LIN {X 0,Y 246.897,Z 628.128,A -85,B 0,C 180,E1 -18808.369,E2 -18808.369} C_VEL
LIN {X 0,Y 246.935,Z 628.341,A -85,B 0,C 180,E1 -18810,E2 -18810} C_VEL
LIN {X 0,Y 246.897,Z 628.119,A -85,B 0,C 180,E1 -18811.631,E2 -18811.631} C_VEL
LIN {X 0,Y 246.851,Z 627.504,A -85,B 0,C 180,E1 -18813.264,E2 -18813.264} C_VEL
LIN {X 0,Y 246.882,Z 626.502,A -85,B 0,C 180,E1 -18814.899,E2 -18814.899} C_VEL
LIN {X 0,Y 247.009,Z 625.098,A -85,B 0,C 180,E1 -18816.535,E2 -18816.535} C_VEL
LIN {X 0,Y 247.457,Z 622.154,A -85,B 0,C 180,E1 -18818.986,E2 -18818.986} C_VEL
LIN {X 0,Y 248.175,Z 618.171,A -85,B 0,C 180,E1 -18821.433,E2 -18821.433} C_VEL
LIN {X 0,Y 249.492,Z 612.051,A -85,B 0,C 180,E1 -18824.269,E2 -18824.269} C_VEL
LIN {X 0,Y 251.197,Z 605.373,A -85,B 0,C 180,E1 -18826.665,E2 -18826.665} C_VEL
LIN {X 0,Y 253.135,Z 596.963,A -85,B 0,C 180,E1 -18829.074,E2 -18829.074} C_VEL
LIN {X 0,Y 254.923,Z 588.585,A -85,B 0,C 180,E1 -18831.002,E2 -18831.002} C_VEL
LIN {X 0,Y 257.208,Z 578.088,A -85,B 0,C 180,E1 -18832.915,E2 -18832.915} C_VEL
LIN {X 0,Y 259.508,Z 566.272,A -85,B 0,C 180,E1 -18834.606,E2 -18834.606} C_VEL
LIN {X 0,Y 261.51,Z 554.368,A -85,B 0,C 180,E1 -18835.894,E2 -18835.894} C_VEL
LIN {X 0,Y 263.118,Z 541.975,A -85,B 0,C 180,E1 -18836.898,E2 -18836.898} C_VEL
LIN {X 0,Y 264.477,Z 529.21,A -85,B 0,C 180,E1 -18837.605,E2 -18837.605} C_VEL
LIN {X 0,Y 265.172,Z 515.69,A -85,B 0,C 180,E1 -18838.063,E2 -18838.063} C_VEL
LIN {X 0,Y 266.746,Z 464.43,A -85,B 0,C 180,E1 -18839.422,E2 -18839.422} C_VEL
LIN {X 0,Y 263.377,Z 442.333,A -85,B 0,C 180,E1 -18840.514,E2 -18840.514} C_VEL
LIN {X 0,Y 259.763,Z 432.973,A -85,B 0,C 180,E1 -18841.277,E2 -18841.277} C_VEL
LIN {X 0,Y 253.442,Z 418.863,A -85,B 0,C 180,E1 -18842.606,E2 -18842.606} C_VEL
LIN {X 0,Y 252.141,Z 415.736,A -85,B 0,C 180,E1 -18842.927,E2 -18842.927} C_VEL
LIN {X 0,Y 250.111,Z 407.153,A -85,B 0,C 180,E1 -18846.663,E2 -18846.663} C_VEL
LIN {X 0,Y 249.039,Z 402.966,A -85,B 0,C 180,E1 -18848.636,E2 -18848.636} C_VEL
LIN {X 0,Y 249.012,Z 402.968,A -85,B 0,C 180,E1 -18852.793,E2 -18852.793} C_VEL
LIN {X 0,Y 249.019,Z 402.965,A -85,B 0,C 180,E1 -18857.363,E2 -18857.363} C_VEL
LIN {X 0,Y 249.044,Z 402.958,A -85,B 0,C 180,E1 -18862.2,E2 -18862.2} C_VEL
LIN {X 0,Y 249.044,Z 402.958,A -85,B 0,C 180,E1 -18865.639,E2 -18865.639} C_VEL
LIN {X 0,Y 249.048,Z 402.96,A -85,B 0,C 180,E1 -18869.473,E2 -18869.473} C_VEL
LIN {X 0,Y 249.073,Z 402.959,A -85,B 0,C 180,E1 -18873.162,E2 -18873.162} C_VEL
LIN {X 0,Y 249.086,Z 402.955,A -85,B 0,C 180,E1 -18876.733,E2 -18876.733} C_VEL
LIN {X 0,Y 249.131,Z 402.949,A -85,B 0,C 180,E1 -18880.213,E2 -18880.213} C_VEL
LIN {X 0,Y 249.243,Z 402.937,A -85,B 0,C 180,E1 -18883.622,E2 -18883.622} C_VEL
LIN {X 0,Y 249.247,Z 402.936,A -85,B 0,C 180,E1 -18888.616,E2 -18888.616} C_VEL
LIN {X 0,Y 249.448,Z 402.91,A -85,B 0,C 180,E1 -18891.902,E2 -18891.902} C_VEL
LIN {X 0,Y 249.296,Z 402.924,A -85,B 0,C 180,E1 -18895.149,E2 -18895.149} C_VEL
LIN {X 0,Y 249.677,Z 402.885,A -85,B 0,C 180,E1 -18898.387,E2 -18898.387} C_VEL
LIN {X 0,Y 249.679,Z 402.876,A -85,B 0,C 180,E1 -18901.613,E2 -18901.613} C_VEL
LIN {X 0,Y 249.454,Z 402.905,A -85,B 0,C 180,E1 -18906.752,E2 -18906.752} C_VEL
LIN {X 0,Y 249.426,Z 402.916,A -85,B 0,C 180,E1 -18909.733,E2 -18909.733} C_VEL
LIN {X 0,Y 249.208,Z 402.941,A -85,B 0,C 180,E1 -18914.703,E2 -18914.703} C_VEL
LIN {X 0,Y 249.143,Z 402.948,A -85,B 0,C 180,E1 -18918.077,E2 -18918.077} C_VEL
LIN {X 0,Y 249.106,Z 402.951,A -85,B 0,C 180,E1 -18921.517,E2 -18921.517} C_VEL
LIN {X 0,Y 249.132,Z 402.951,A -85,B 0,C 180,E1 -18925.482,E2 -18925.482} C_VEL
LIN {X 0,Y 249.085,Z 402.957,A -85,B 0,C 180,E1 -18928.994,E2 -18928.994} C_VEL
LIN {X 0,Y 249.038,Z 402.962,A -85,B 0,C 180,E1 -18932.425,E2 -18932.425} C_VEL
LIN {X 0,Y 249.076,Z 402.957,A -85,B 0,C 180,E1 -18936.338,E2 -18936.338} C_VEL
LIN {X 0,Y 249.035,Z 402.96,A -85,B 0,C 180,E1 -18940.473,E2 -18940.473} C_VEL
LIN {X 0,Y 248.997,Z 402.966,A -85,B 0,C 180,E1 -18944.881,E2 -18944.881} C_VEL
LIN {X 0,Y 249.011,Z 402.965,A -85,B 0,C 180,E1 -18947.362,E2 -18947.362} C_VEL
LIN {X 0,Y 249.027,Z 402.964,A -85,B 0,C 180,E1 -18951.62,E2 -18951.62} C_VEL
LIN {X 0,Y 249.085,Z 403.063,A -85,B 0,C 180,E1 -18955.283,E2 -18955.283} C_VEL
LIN {X 0,Y 249.966,Z 406.53,A -85,B 0,C 180,E1 -18956.849,E2 -18956.849} C_VEL
LIN {X 0,Y 259.579,Z 426.19,A -85,B 0,C 180,E1 -18958.86,E2 -18958.86} C_VEL
LIN {X 0,Y 265.501,Z 440.501,A -85,B 0,C 180,E1 -18960.074,E2 -18960.074} C_VEL
LIN {X 0,Y 267.41,Z 445.672,A -85,B 0,C 180,E1 -18960.467,E2 -18960.467} C_VEL
LIN {X 0,Y 265.529,Z 503.163,A -85,B 0,C 180,E1 -18961.978,E2 -18961.978} C_VEL
LIN {X 0,Y 264.914,Z 517.263,A -85,B 0,C 180,E1 -18962.445,E2 -18962.445} C_VEL
LIN {X 0,Y 263.654,Z 530.366,A -85,B 0,C 180,E1 -18963.161,E2 -18963.161} C_VEL
LIN {X 0,Y 262.194,Z 542.855,A -85,B 0,C 180,E1 -18964.178,E2 -18964.178} C_VEL
LIN {X 0,Y 260.317,Z 554.829,A -85,B 0,C 180,E1 -18965.475,E2 -18965.475} C_VEL
LIN {X 0,Y 258.34,Z 565.491,A -85,B 0,C 180,E1 -18966.979,E2 -18966.979} C_VEL
LIN {X 0,Y 256.193,Z 576.011,A -85,B 0,C 180,E1 -18968.861,E2 -18968.861} C_VEL
LIN {X 0,Y 254.115,Z 585.636,A -85,B 0,C 180,E1 -18971.037,E2 -18971.037} C_VEL
LIN {X 0,Y 251.998,Z 593.891,A -85,B 0,C 180,E1 -18973.39,E2 -18973.39} C_VEL
LIN {X 0,Y 250.403,Z 600.535,A -85,B 0,C 180,E1 -18975.784,E2 -18975.784} C_VEL
LIN {X 0,Y 248.88,Z 606.622,A -85,B 0,C 180,E1 -18978.6,E2 -18978.6} C_VEL
LIN {X 0,Y 247.984,Z 610.573,A -85,B 0,C 180,E1 -18981.033,E2 -18981.033} C_VEL
LIN {X 0,Y 247.27,Z 614.095,A -85,B 0,C 180,E1 -18984.147,E2 -18984.147} C_VEL
LIN {X 0,Y 247.072,Z 615.873,A -85,B 0,C 180,E1 -18986.739,E2 -18986.739} C_VEL
LIN {X 0,Y 246.943,Z 616.713,A -85,B 0,C 180,E1 -18990,E2 -18990} C_VEL
LIN {X 0,Y 246.97,Z 616.519,A -85,B 0,C 180,E1 -18991.631,E2 -18991.631} C_VEL
LIN {X 0,Y 247.071,Z 615.932,A -85,B 0,C 180,E1 -18993.262,E2 -18993.262} C_VEL
LIN {X 0,Y 247.394,Z 613.607,A -85,B 0,C 180,E1 -18996.525,E2 -18996.525} C_VEL
LIN {X 0,Y 248.008,Z 610.735,A -85,B 0,C 180,E1 -18998.967,E2 -18998.967} C_VEL
LIN {X 0,Y 248.855,Z 606.842,A -85,B 0,C 180,E1 -19001.402,E2 -19001.402} C_VEL
LIN {X 0,Y 250.068,Z 601.817,A -85,B 0,C 180,E1 -19003.821,E2 -19003.821} C_VEL
LIN {X 0,Y 251.638,Z 595.488,A -85,B 0,C 180,E1 -19006.218,E2 -19006.218} C_VEL
LIN {X 0,Y 253.672,Z 587.566,A -85,B 0,C 180,E1 -19008.579,E2 -19008.579} C_VEL
LIN {X 0,Y 255.549,Z 579.262,A -85,B 0,C 180,E1 -19010.582,E2 -19010.582} C_VEL
LIN {X 0,Y 257.507,Z 569.641,A -85,B 0,C 180,E1 -19012.464,E2 -19012.464} C_VEL
LIN {X 0,Y 259.466,Z 559.937,A -85,B 0,C 180,E1 -19013.973,E2 -19013.973} C_VEL
LIN {X 0,Y 261.312,Z 549.424,A -85,B 0,C 180,E1 -19015.275,E2 -19015.275} C_VEL
LIN {X 0,Y 263.028,Z 536.765,A -85,B 0,C 180,E1 -19016.48,E2 -19016.48} C_VEL
LIN {X 0,Y 264.376,Z 524.073,A -85,B 0,C 180,E1 -19017.348,E2 -19017.348} C_VEL
LIN {X 0,Y 265.3,Z 511.903,A -85,B 0,C 180,E1 -19017.887,E2 -19017.887} C_VEL
LIN {X 0,Y 267.516,Z 446.684,A -85,B 0,C 180,E1 -19019.619,E2 -19019.619} C_VEL
LIN {X 0,Y 266.944,Z 444.324,A -85,B 0,C 180,E1 -19019.761,E2 -19019.761} C_VEL
LIN {X 0,Y 260.106,Z 427.321,A -85,B 0,C 180,E1 -19021.168,E2 -19021.168} C_VEL
LIN {X 0,Y 253.049,Z 412.735,A -85,B 0,C 180,E1 -19022.626,E2 -19022.626} C_VEL
LIN {X 0,Y 249.84,Z 406.254,A -85,B 0,C 180,E1 -19023.325,E2 -19023.325} C_VEL
LIN {X 0,Y 249.074,Z 402.959,A -85,B 0,C 180,E1 -19024.946,E2 -19024.946} C_VEL
LIN {X 0,Y 249.029,Z 402.966,A -85,B 0,C 180,E1 -19028.381,E2 -19028.381} C_VEL
LIN {X 0,Y 249.015,Z 402.965,A -85,B 0,C 180,E1 -19032.793,E2 -19032.793} C_VEL
LIN {X 0,Y 249.031,Z 402.964,A -85,B 0,C 180,E1 -19037.366,E2 -19037.366} C_VEL
LIN {X 0,Y 249.051,Z 402.951,A -85,B 0,C 180,E1 -19041.624,E2 -19041.624} C_VEL
LIN {X 0,Y 249.065,Z 402.957,A -85,B 0,C 180,E1 -19045.643,E2 -19045.643} C_VEL
LIN {X 0,Y 249.056,Z 402.959,A -85,B 0,C 180,E1 -19049.473,E2 -19049.473} C_VEL
LIN {X 0,Y 249.078,Z 402.957,A -85,B 0,C 180,E1 -19053.163,E2 -19053.163} C_VEL
LIN {X 0,Y 249.089,Z 402.957,A -85,B 0,C 180,E1 -19056.733,E2 -19056.733} C_VEL
LIN {X 0,Y 249.134,Z 402.945,A -85,B 0,C 180,E1 -19060.213,E2 -19060.213} C_VEL
LIN {X 0,Y 249.246,Z 402.938,A -85,B 0,C 180,E1 -19063.622,E2 -19063.622} C_VEL
LIN {X 0,Y 249.257,Z 402.935,A -85,B 0,C 180,E1 -19068.617,E2 -19068.617} C_VEL
LIN {X 0,Y 249.489,Z 402.9,A -85,B 0,C 180,E1 -19071.903,E2 -19071.903} C_VEL
LIN {X 0,Y 249.441,Z 402.911,A -85,B 0,C 180,E1 -19076.77,E2 -19076.77} C_VEL
LIN {X 0,Y 249.732,Z 402.87,A -85,B 0,C 180,E1 -19080,E2 -19080} C_VEL
LIN {X 0,Y 249.44,Z 402.913,A -85,B 0,C 180,E1 -19083.23,E2 -19083.23} C_VEL
LIN {X 0,Y 249.379,Z 402.913,A -85,B 0,C 180,E1 -19085.93,E2 -19085.93} C_VEL
LIN {X 0,Y 248.793,Z 402.992,A -85,B 0,C 180,E1 -19087.278,E2 -19087.278} C_VEL
LIN {X 0,Y 247.186,Z 403.196,A -85,B 0,C 180,E1 -19088.599,E2 -19088.599} C_VEL
LIN {X 0,Y 243.308,Z 403.67,A -85,B 0,C 180,E1 -19091.256,E2 -19091.256} C_VEL
LIN {X 0,Y 242.232,Z 403.806,A -85,B 0,C 180,E1 -19092.646,E2 -19092.646} C_VEL
LIN {X 0,Y 242.158,Z 403.815,A -85,B 0,C 180,E1 -19093.118,E2 -19093.118} C_VEL
LIN {X 0,Y 242.154,Z 403.814,A -85,B 0,C 180,E1 -19096.872,E2 -19096.872} C_VEL
LIN {X 0,Y 242.057,Z 403.827,A -85,B 0,C 180,E1 -19101.703,E2 -19101.703} C_VEL
LIN {X 0,Y 242.07,Z 403.831,A -85,B 0,C 180,E1 -19105.838,E2 -19105.838} C_VEL
LIN {X 0,Y 242.01,Z 403.839,A -85,B 0,C 180,E1 -19109.583,E2 -19109.583} C_VEL
LIN {X 0,Y 241.983,Z 403.842,A -85,B 0,C 180,E1 -19113.492,E2 -19113.492} C_VEL
LIN {X 0,Y 241.989,Z 403.84,A -85,B 0,C 180,E1 -19117.582,E2 -19117.582} C_VEL
LIN {X 0,Y 241.942,Z 403.847,A -85,B 0,C 180,E1 -19121.922,E2 -19121.922} C_VEL
LIN {X 0,Y 241.939,Z 403.848,A -85,B 0,C 180,E1 -19126.57,E2 -19126.57} C_VEL
LIN {X 0,Y 242.019,Z 404.013,A -85,B 0,C 180,E1 -19130.569,E2 -19130.569} C_VEL
LIN {X 0,Y 243.966,Z 411.663,A -85,B 0,C 180,E1 -19134.173,E2 -19134.173} C_VEL
LIN {X 0,Y 244.982,Z 415.904,A -85,B 0,C 180,E1 -19135.975,E2 -19135.975} C_VEL
LIN {X 0,Y 253.639,Z 434.761,A -85,B 0,C 180,E1 -19137.897,E2 -19137.897} C_VEL
LIN {X 0,Y 257.526,Z 444.708,A -85,B 0,C 180,E1 -19138.753,E2 -19138.753} C_VEL
LIN {X 0,Y 260.655,Z 464.974,A -85,B 0,C 180,E1 -19139.801,E2 -19139.801} C_VEL
LIN {X 0,Y 258.602,Z 524.234,A -85,B 0,C 180,E1 -19141.435,E2 -19141.435} C_VEL
LIN {X 0,Y 257.39,Z 537.372,A -85,B 0,C 180,E1 -19142.066,E2 -19142.066} C_VEL
LIN {X 0,Y 255.941,Z 549.464,A -85,B 0,C 180,E1 -19142.948,E2 -19142.948} C_VEL
LIN {X 0,Y 253.941,Z 561.67,A -85,B 0,C 180,E1 -19144.157,E2 -19144.157} C_VEL
LIN {X 0,Y 251.743,Z 573.234,A -85,B 0,C 180,E1 -19145.683,E2 -19145.683} C_VEL
LIN {X 0,Y 249.428,Z 583.648,A -85,B 0,C 180,E1 -19147.424,E2 -19147.424} C_VEL
LIN {X 0,Y 247.464,Z 592.165,A -85,B 0,C 180,E1 -19149.206,E2 -19149.206} C_VEL
LIN {X 0,Y 245.617,Z 600.353,A -85,B 0,C 180,E1 -19151.321,E2 -19151.321} C_VEL
LIN {X 0,Y 243.763,Z 607.705,A -85,B 0,C 180,E1 -19153.673,E2 -19153.673} C_VEL
LIN {X 0,Y 241.877,Z 614.785,A -85,B 0,C 180,E1 -19156.558,E2 -19156.558} C_VEL
LIN {X 0,Y 240.89,Z 619.5,A -85,B 0,C 180,E1 -19159.068,E2 -19159.068} C_VEL
LIN {X 0,Y 240.222,Z 623.103,A -85,B 0,C 180,E1 -19161.588,E2 -19161.588} C_VEL
LIN {X 0,Y 239.953,Z 624.961,A -85,B 0,C 180,E1 -19163.272,E2 -19163.272} C_VEL
LIN {X 0,Y 239.755,Z 627.352,A -85,B 0,C 180,E1 -19166.639,E2 -19166.639} C_VEL
LIN {X 0,Y 239.809,Z 627.961,A -85,B 0,C 180,E1 -19168.32,E2 -19168.32} C_VEL
LIN {X 0,Y 239.846,Z 628.174,A -85,B 0,C 180,E1 -19170,E2 -19170} C_VEL
LIN {X 0,Y 239.809,Z 627.951,A -85,B 0,C 180,E1 -19171.679,E2 -19171.679} C_VEL
LIN {X 0,Y 239.771,Z 626.542,A -85,B 0,C 180,E1 -19174.736,E2 -19174.736} C_VEL
LIN {X 0,Y 239.952,Z 624.93,A -85,B 0,C 180,E1 -19176.728,E2 -19176.728} C_VEL
LIN {X 0,Y 240.416,Z 621.985,A -85,B 0,C 180,E1 -19179.252,E2 -19179.252} C_VEL
LIN {X 0,Y 241.198,Z 618.003,A -85,B 0,C 180,E1 -19181.769,E2 -19181.769} C_VEL
LIN {X 0,Y 242.611,Z 611.882,A -85,B 0,C 180,E1 -19184.683,E2 -19184.683} C_VEL
LIN {X 0,Y 244.359,Z 605.203,A -85,B 0,C 180,E1 -19187.145,E2 -19187.145} C_VEL
LIN {X 0,Y 246.242,Z 597.458,A -85,B 0,C 180,E1 -19189.436,E2 -19189.436} C_VEL
LIN {X 0,Y 248.275,Z 588.414,A -85,B 0,C 180,E1 -19191.592,E2 -19191.592} C_VEL
LIN {X 0,Y 250.665,Z 577.917,A -85,B 0,C 180,E1 -19193.549,E2 -19193.549} C_VEL
LIN {X 0,Y 253.059,Z 566.1,A -85,B 0,C 180,E1 -19195.277,E2 -19195.277} C_VEL
LIN {X 0,Y 255.149,Z 554.195,A -85,B 0,C 180,E1 -19196.59,E2 -19196.59} C_VEL
LIN {X 0,Y 256.823,Z 541.801,A -85,B 0,C 180,E1 -19197.613,E2 -19197.613} C_VEL
LIN {X 0,Y 258.22,Z 529.031,A -85,B 0,C 180,E1 -19198.333,E2 -19198.333} C_VEL
LIN {X 0,Y 258.939,Z 515.502,A -85,B 0,C 180,E1 -19198.8,E2 -19198.8} C_VEL
LIN {X 0,Y 260.581,Z 465.599,A -85,B 0,C 180,E1 -19200.147,E2 -19200.147} C_VEL
LIN {X 0,Y 257.439,Z 444.492,A -85,B 0,C 180,E1 -19201.222,E2 -19201.222} C_VEL
LIN {X 0,Y 251.429,Z 429.81,A -85,B 0,C 180,E1 -19202.534,E2 -19202.534} C_VEL
LIN {X 0,Y 246.214,Z 418.717,A -85,B 0,C 180,E1 -19203.685,E2 -19203.685} C_VEL
LIN {X 0,Y 244.856,Z 415.514,A -85,B 0,C 180,E1 -19204.047,E2 -19204.047} C_VEL
LIN {X 0,Y 242.907,Z 407.421,A -85,B 0,C 180,E1 -19207.738,E2 -19207.738} C_VEL
LIN {X 0,Y 241.986,Z 403.841,A -85,B 0,C 180,E1 -19209.531,E2 -19209.531} C_VEL
LIN {X 0,Y 241.935,Z 403.845,A -85,B 0,C 180,E1 -19214.201,E2 -19214.201} C_VEL
LIN {X 0,Y 241.94,Z 403.846,A -85,B 0,C 180,E1 -19218.078,E2 -19218.078} C_VEL
LIN {X 0,Y 241.99,Z 403.836,A -85,B 0,C 180,E1 -19222.418,E2 -19222.418} C_VEL
LIN {X 0,Y 241.981,Z 403.841,A -85,B 0,C 180,E1 -19226.507,E2 -19226.507} C_VEL
LIN {X 0,Y 242.014,Z 403.84,A -85,B 0,C 180,E1 -19230.597,E2 -19230.597} C_VEL
LIN {X 0,Y 242.069,Z 403.832,A -85,B 0,C 180,E1 -19234.183,E2 -19234.183} C_VEL
LIN {X 0,Y 242.066,Z 403.833,A -85,B 0,C 180,E1 -19238.29,E2 -19238.29} C_VEL
LIN {X 0,Y 242.164,Z 403.819,A -85,B 0,C 180,E1 -19243.278,E2 -19243.278} C_VEL
LIN {X 0,Y 242.183,Z 403.819,A -85,B 0,C 180,E1 -19248.28,E2 -19248.28} C_VEL
LIN {X 0,Y 242.395,Z 403.788,A -85,B 0,C 180,E1 -19251.665,E2 -19251.665} C_VEL
LIN {X 0,Y 242.257,Z 403.801,A -85,B 0,C 180,E1 -19255.007,E2 -19255.007} C_VEL
LIN {X 0,Y 242.638,Z 403.762,A -85,B 0,C 180,E1 -19258.34,E2 -19258.34} C_VEL
LIN {X 0,Y 242.639,Z 403.753,A -85,B 0,C 180,E1 -19261.66,E2 -19261.66} C_VEL
LIN {X 0,Y 242.432,Z 403.78,A -85,B 0,C 180,E1 -19266.731,E2 -19266.731} C_VEL
LIN {X 0,Y 242.347,Z 403.797,A -85,B 0,C 180,E1 -19270.02,E2 -19270.02} C_VEL
LIN {X 0,Y 242.169,Z 403.818,A -85,B 0,C 180,E1 -19275.141,E2 -19275.141} C_VEL
LIN {X 0,Y 242.082,Z 403.829,A -85,B 0,C 180,E1 -19278.624,E2 -19278.624} C_VEL
LIN {X 0,Y 242.052,Z 403.83,A -85,B 0,C 180,E1 -19282.176,E2 -19282.176} C_VEL
LIN {X 0,Y 242.068,Z 403.828,A -85,B 0,C 180,E1 -19285.838,E2 -19285.838} C_VEL
LIN {X 0,Y 242.032,Z 403.834,A -85,B 0,C 180,E1 -19289.58,E2 -19289.58} C_VEL
LIN {X 0,Y 241.993,Z 403.839,A -85,B 0,C 180,E1 -19293.491,E2 -19293.491} C_VEL
LIN {X 0,Y 242.012,Z 403.835,A -85,B 0,C 180,E1 -19297.578,E2 -19297.578} C_VEL
LIN {X 0,Y 241.95,Z 403.846,A -85,B 0,C 180,E1 -19301.92,E2 -19301.92} C_VEL
LIN {X 0,Y 241.928,Z 403.847,A -85,B 0,C 180,E1 -19306.573,E2 -19306.573} C_VEL
LIN {X 0,Y 241.958,Z 403.846,A -85,B 0,C 180,E1 -19310.281,E2 -19310.281} C_VEL
LIN {X 0,Y 242.03,Z 403.853,A -85,B 0,C 180,E1 -19314.396,E2 -19314.396} C_VEL
LIN {X 0,Y 242.707,Z 406.604,A -85,B 0,C 180,E1 -19315.716,E2 -19315.716} C_VEL
LIN {X 0,Y 251.706,Z 424.526,A -85,B 0,C 180,E1 -19317.707,E2 -19317.707} C_VEL
LIN {X 0,Y 257.992,Z 438.988,A -85,B 0,C 180,E1 -19319.053,E2 -19319.053} C_VEL
LIN {X 0,Y 261.168,Z 447.286,A -85,B 0,C 180,E1 -19319.733,E2 -19319.733} C_VEL
LIN {X 0,Y 259.33,Z 502.465,A -85,B 0,C 180,E1 -19321.219,E2 -19321.219} C_VEL
LIN {X 0,Y 258.621,Z 517.764,A -85,B 0,C 180,E1 -19321.73,E2 -19321.73} C_VEL
LIN {X 0,Y 257.351,Z 530.542,A -85,B 0,C 180,E1 -19322.449,E2 -19322.449} C_VEL
LIN {X 0,Y 255.835,Z 543.028,A -85,B 0,C 180,E1 -19323.487,E2 -19323.487} C_VEL
LIN {X 0,Y 253.894,Z 555.001,A -85,B 0,C 180,E1 -19324.812,E2 -19324.812} C_VEL
LIN {X 0,Y 251.82,Z 565.662,A -85,B 0,C 180,E1 -19326.348,E2 -19326.348} C_VEL
LIN {X 0,Y 249.461,Z 576.75,A -85,B 0,C 180,E1 -19328.389,E2 -19328.389} C_VEL
LIN {X 0,Y 247.413,Z 585.805,A -85,B 0,C 180,E1 -19330.502,E2 -19330.502} C_VEL
LIN {X 0,Y 245.206,Z 594.06,A -85,B 0,C 180,E1 -19332.916,E2 -19332.916} C_VEL
LIN {X 0,Y 243.523,Z 600.704,A -85,B 0,C 180,E1 -19335.373,E2 -19335.373} C_VEL
LIN {X 0,Y 241.921,Z 606.791,A -85,B 0,C 180,E1 -19338.267,E2 -19338.267} C_VEL
LIN {X 0,Y 240.972,Z 610.741,A -85,B 0,C 180,E1 -19340.77,E2 -19340.77} C_VEL
LIN {X 0,Y 240.171,Z 614.479,A -85,B 0,C 180,E1 -19344.227,E2 -19344.227} C_VEL
LIN {X 0,Y 239.995,Z 616.04,A -85,B 0,C 180,E1 -19346.643,E2 -19346.643} C_VEL
LIN {X 0,Y 239.885,Z 616.65,A -85,B 0,C 180,E1 -19348.321,E2 -19348.321} C_VEL
LIN {X 0,Y 239.854,Z 616.88,A -85,B 0,C 180,E1 -19350,E2 -19350} C_VEL
LIN {X 0,Y 239.885,Z 616.686,A -85,B 0,C 180,E1 -19351.679,E2 -19351.679} C_VEL
LIN {X 0,Y 239.994,Z 616.099,A -85,B 0,C 180,E1 -19353.358,E2 -19353.358} C_VEL
LIN {X 0,Y 240.349,Z 613.773,A -85,B 0,C 180,E1 -19356.717,E2 -19356.717} C_VEL
LIN {X 0,Y 240.988,Z 610.902,A -85,B 0,C 180,E1 -19359.23,E2 -19359.23} C_VEL
LIN {X 0,Y 241.893,Z 607.008,A -85,B 0,C 180,E1 -19361.735,E2 -19361.735} C_VEL
LIN {X 0,Y 243.176,Z 601.983,A -85,B 0,C 180,E1 -19364.221,E2 -19364.221} C_VEL
LIN {X 0,Y 244.825,Z 595.654,A -85,B 0,C 180,E1 -19366.683,E2 -19366.683} C_VEL
LIN {X 0,Y 246.957,Z 587.731,A -85,B 0,C 180,E1 -19369.104,E2 -19369.104} C_VEL
LIN {X 0,Y 248.766,Z 580.035,A -85,B 0,C 180,E1 -19371.021,E2 -19371.021} C_VEL
LIN {X 0,Y 250.962,Z 569.804,A -85,B 0,C 180,E1 -19373.083,E2 -19373.083} C_VEL
LIN {X 0,Y 253.282,Z 558.705,A -85,B 0,C 180,E1 -19374.815,E2 -19374.815} C_VEL
LIN {X 0,Y 255.181,Z 547.823,A -85,B 0,C 180,E1 -19376.146,E2 -19376.146} C_VEL
LIN {X 0,Y 256.851,Z 535.797,A -85,B 0,C 180,E1 -19377.279,E2 -19377.279} C_VEL
LIN {X 0,Y 258.152,Z 523.418,A -85,B 0,C 180,E1 -19378.121,E2 -19378.121} C_VEL
LIN {X 0,Y 259.07,Z 510.548,A -85,B 0,C 180,E1 -19378.674,E2 -19378.674} C_VEL
LIN {X 0,Y 259.842,Z 490.019,A -85,B 0,C 180,E1 -19379.236,E2 -19379.236} C_VEL
LIN {X 0,Y 261.259,Z 447.451,A -85,B 0,C 180,E1 -19380.383,E2 -19380.383} C_VEL
LIN {X 0,Y 255.083,Z 431.858,A -85,B 0,C 180,E1 -19381.709,E2 -19381.709} C_VEL
LIN {X 0,Y 248.25,Z 417.405,A -85,B 0,C 180,E1 -19383.183,E2 -19383.183} C_VEL
LIN {X 0,Y 242.656,Z 406.378,A -85,B 0,C 180,E1 -19384.479,E2 -19384.479} C_VEL
LIN {X 0,Y 242.009,Z 403.833,A -85,B 0,C 180,E1 -19385.808,E2 -19385.808} C_VEL
LIN {X 0,Y 241.959,Z 403.846,A -85,B 0,C 180,E1 -19389.719,E2 -19389.719} C_VEL
LIN {X 0,Y 241.939,Z 403.848,A -85,B 0,C 180,E1 -19394.201,E2 -19394.201} C_VEL
LIN {X 0,Y 241.956,Z 403.844,A -85,B 0,C 180,E1 -19398.081,E2 -19398.081} C_VEL
LIN {X 0,Y 242.014,Z 403.831,A -85,B 0,C 180,E1 -19402.422,E2 -19402.422} C_VEL
LIN {X 0,Y 241.995,Z 403.837,A -85,B 0,C 180,E1 -19406.509,E2 -19406.509} C_VEL
LIN {X 0,Y 242.041,Z 403.83,A -85,B 0,C 180,E1 -19410.587,E2 -19410.587} C_VEL
LIN {X 0,Y 242.071,Z 403.827,A -85,B 0,C 180,E1 -19414.183,E2 -19414.183} C_VEL
LIN {X 0,Y 242.069,Z 403.832,A -85,B 0,C 180,E1 -19418.29,E2 -19418.29} C_VEL
LIN {X 0,Y 242.167,Z 403.818,A -85,B 0,C 180,E1 -19423.278,E2 -19423.278} C_VEL
LIN {X 0,Y 242.191,Z 403.815,A -85,B 0,C 180,E1 -19428.28,E2 -19428.28} C_VEL
LIN {X 0,Y 242.44,Z 403.78,A -85,B 0,C 180,E1 -19431.666,E2 -19431.666} C_VEL
LIN {X 0,Y 242.266,Z 403.805,A -85,B 0,C 180,E1 -19435.007,E2 -19435.007} C_VEL
LIN {X 0,Y 242.641,Z 403.751,A -85,B 0,C 180,E1 -19438.34,E2 -19438.34} C_VEL
LIN {X 0,Y 242.641,Z 403.76,A -85,B 0,C 180,E1 -19441.66,E2 -19441.66} C_VEL
LIN {X 0,Y 242.422,Z 403.782,A -85,B 0,C 180,E1 -19446.659,E2 -19446.659} C_VEL
LIN {X 0,Y 242.271,Z 403.802,A -85,B 0,C 180,E1 -19450.023,E2 -19450.023} C_VEL
LIN {X 0,Y 242.158,Z 403.815,A -85,B 0,C 180,E1 -19453.118,E2 -19453.118} C_VEL
LIN {X 0,Y 241.506,Z 403.904,A -85,B 0,C 180,E1 -19454.506,E2 -19454.506} C_VEL
LIN {X 0,Y 238.588,Z 404.266,A -85,B 0,C 180,E1 -19456.766,E2 -19456.766} C_VEL
LIN {X 0,Y 236.104,Z 404.571,A -85,B 0,C 180,E1 -19458.609,E2 -19458.609} C_VEL
LIN {X 0,Y 235.062,Z 404.704,A -85,B 0,C 180,E1 -19460.041,E2 -19460.041} C_VEL
LIN {X 0,Y 234.991,Z 404.71,A -85,B 0,C 180,E1 -19460.527,E2 -19460.527} C_VEL
LIN {X 0,Y 234.991,Z 404.713,A -85,B 0,C 180,E1 -19464.753,E2 -19464.753} C_VEL
LIN {X 0,Y 234.94,Z 404.717,A -85,B 0,C 180,E1 -19468.596,E2 -19468.596} C_VEL
LIN {X 0,Y 234.946,Z 404.718,A -85,B 0,C 180,E1 -19473.114,E2 -19473.114} C_VEL
LIN {X 0,Y 234.928,Z 404.719,A -85,B 0,C 180,E1 -19476.749,E2 -19476.749} C_VEL
LIN {X 0,Y 234.944,Z 404.718,A -85,B 0,C 180,E1 -19478.944,E2 -19478.944} C_VEL
LIN {X 0,Y 234.892,Z 404.726,A -85,B 0,C 180,E1 -19483.485,E2 -19483.485} C_VEL
LIN {X 0,Y 234.892,Z 404.726,A -85,B 0,C 180,E1 -19486.514,E2 -19486.514} C_VEL
LIN {X 0,Y 234.923,Z 404.875,A -85,B 0,C 180,E1 -19489.619,E2 -19489.619} C_VEL
LIN {X 0,Y 237.05,Z 413.026,A -85,B 0,C 180,E1 -19493.632,E2 -19493.632} C_VEL
LIN {X 0,Y 237.559,Z 415.398,A -85,B 0,C 180,E1 -19494.734,E2 -19494.734} C_VEL
LIN {X 0,Y 239.563,Z 419.492,A -85,B 0,C 180,E1 -19495.228,E2 -19495.228} C_VEL
LIN {X 0,Y 247.265,Z 436.042,A -85,B 0,C 180,E1 -19497.014,E2 -19497.014} C_VEL
LIN {X 0,Y 251.734,Z 447.593,A -85,B 0,C 180,E1 -19498.049,E2 -19498.049} C_VEL
LIN {X 0,Y 254.565,Z 466.785,A -85,B 0,C 180,E1 -19499.063,E2 -19499.063} C_VEL
LIN {X 0,Y 252.388,Z 524.081,A -85,B 0,C 180,E1 -19500.664,E2 -19500.664} C_VEL
LIN {X 0,Y 251.157,Z 537.215,A -85,B 0,C 180,E1 -19501.309,E2 -19501.309} C_VEL
LIN {X 0,Y 249.643,Z 549.304,A -85,B 0,C 180,E1 -19502.207,E2 -19502.207} C_VEL
LIN {X 0,Y 247.574,Z 561.507,A -85,B 0,C 180,E1 -19503.441,E2 -19503.441} C_VEL
LIN {X 0,Y 245.257,Z 573.07,A -85,B 0,C 180,E1 -19504.996,E2 -19504.996} C_VEL
LIN {X 0,Y 242.889,Z 583.484,A -85,B 0,C 180,E1 -19506.781,E2 -19506.781} C_VEL
LIN {X 0,Y 240.812,Z 592,A -85,B 0,C 180,E1 -19508.604,E2 -19508.604} C_VEL
LIN {X 0,Y 239.019,Z 599.673,A -85,B 0,C 180,E1 -19510.625,E2 -19510.625} C_VEL
LIN {X 0,Y 236.94,Z 607.539,A -85,B 0,C 180,E1 -19513.19,E2 -19513.19} C_VEL
LIN {X 0,Y 234.938,Z 614.618,A -85,B 0,C 180,E1 -19516.154,E2 -19516.154} C_VEL
LIN {X 0,Y 233.905,Z 619.333,A -85,B 0,C 180,E1 -19518.737,E2 -19518.737} C_VEL
LIN {X 0,Y 233.191,Z 622.936,A -85,B 0,C 180,E1 -19521.333,E2 -19521.333} C_VEL
LIN {X 0,Y 232.89,Z 624.795,A -85,B 0,C 180,E1 -19523.067,E2 -19523.067} C_VEL
LIN {X 0,Y 232.664,Z 627.185,A -85,B 0,C 180,E1 -19526.536,E2 -19526.536} C_VEL
LIN {X 0,Y 232.722,Z 627.795,A -85,B 0,C 180,E1 -19528.269,E2 -19528.269} C_VEL
LIN {X 0,Y 232.759,Z 628.008,A -85,B 0,C 180,E1 -19530,E2 -19530} C_VEL
LIN {X 0,Y 232.722,Z 627.784,A -85,B 0,C 180,E1 -19531.73,E2 -19531.73} C_VEL
LIN {X 0,Y 232.731,Z 626.167,A -85,B 0,C 180,E1 -19535.197,E2 -19535.197} C_VEL
LIN {X 0,Y 232.89,Z 624.762,A -85,B 0,C 180,E1 -19536.933,E2 -19536.933} C_VEL
LIN {X 0,Y 233.395,Z 621.817,A -85,B 0,C 180,E1 -19539.533,E2 -19539.533} C_VEL
LIN {X 0,Y 234.231,Z 617.834,A -85,B 0,C 180,E1 -19542.124,E2 -19542.124} C_VEL
LIN {X 0,Y 235.736,Z 611.713,A -85,B 0,C 180,E1 -19545.121,E2 -19545.121} C_VEL
LIN {X 0,Y 237.519,Z 605.033,A -85,B 0,C 180,E1 -19547.655,E2 -19547.655} C_VEL
LIN {X 0,Y 239.365,Z 597.938,A -85,B 0,C 180,E1 -19549.823,E2 -19549.823} C_VEL
LIN {X 0,Y 241.667,Z 588.244,A -85,B 0,C 180,E1 -19552.213,E2 -19552.213} C_VEL
LIN {X 0,Y 244.172,Z 577.746,A -85,B 0,C 180,E1 -19554.215,E2 -19554.215} C_VEL
LIN {X 0,Y 246.658,Z 565.928,A -85,B 0,C 180,E1 -19555.981,E2 -19555.981} C_VEL
LIN {X 0,Y 248.823,Z 554.022,A -85,B 0,C 180,E1 -19557.321,E2 -19557.321} C_VEL
LIN {X 0,Y 250.38,Z 542.927,A -85,B 0,C 180,E1 -19558.273,E2 -19558.273} C_VEL
LIN {X 0,Y 251.928,Z 529.783,A -85,B 0,C 180,E1 -19559.05,E2 -19559.05} C_VEL
LIN {X 0,Y 252.687,Z 517.104,A -85,B 0,C 180,E1 -19559.525,E2 -19559.525} C_VEL
LIN {X 0,Y 254.357,Z 465.807,A -85,B 0,C 180,E1 -19560.952,E2 -19560.952} C_VEL
LIN {X 0,Y 251.523,Z 446.656,A -85,B 0,C 180,E1 -19561.965,E2 -19561.965} C_VEL
LIN {X 0,Y 244.883,Z 430.758,A -85,B 0,C 180,E1 -19563.477,E2 -19563.477} C_VEL
LIN {X 0,Y 239.172,Z 418.866,A -85,B 0,C 180,E1 -19564.804,E2 -19564.804} C_VEL
LIN {X 0,Y 237.555,Z 415.333,A -85,B 0,C 180,E1 -19565.237,E2 -19565.237} C_VEL
LIN {X 0,Y 235.776,Z 407.971,A -85,B 0,C 180,E1 -19568.753,E2 -19568.753} C_VEL
LIN {X 0,Y 234.913,Z 404.724,A -85,B 0,C 180,E1 -19570.453,E2 -19570.453} C_VEL
LIN {X 0,Y 234.899,Z 404.721,A -85,B 0,C 180,E1 -19574.105,E2 -19574.105} C_VEL
LIN {X 0,Y 234.885,Z 404.722,A -85,B 0,C 180,E1 -19578.832,E2 -19578.832} C_VEL
LIN {X 0,Y 234.919,Z 404.72,A -85,B 0,C 180,E1 -19581.079,E2 -19581.079} C_VEL
LIN {X 0,Y 234.931,Z 404.716,A -85,B 0,C 180,E1 -19585.362,E2 -19585.362} C_VEL
LIN {X 0,Y 234.923,Z 404.72,A -85,B 0,C 180,E1 -19589.431,E2 -19589.431} C_VEL
LIN {X 0,Y 234.995,Z 404.712,A -85,B 0,C 180,E1 -19593.794,E2 -19593.794} C_VEL
LIN {X 0,Y 235.029,Z 404.708,A -85,B 0,C 180,E1 -19598.971,E2 -19598.971} C_VEL
LIN {X 0,Y 235.098,Z 404.699,A -85,B 0,C 180,E1 -19603.059,E2 -19603.059} C_VEL
LIN {X 0,Y 235.117,Z 404.698,A -85,B 0,C 180,E1 -19607.922,E2 -19607.922} C_VEL
LIN {X 0,Y 235.328,Z 404.667,A -85,B 0,C 180,E1 -19611.412,E2 -19611.412} C_VEL
LIN {X 0,Y 235.37,Z 404.665,A -85,B 0,C 180,E1 -19613.14,E2 -19613.14} C_VEL
LIN {X 0,Y 235.597,Z 404.64,A -85,B 0,C 180,E1 -19618.291,E2 -19618.291} C_VEL
LIN {X 0,Y 235.599,Z 404.63,A -85,B 0,C 180,E1 -19621.709,E2 -19621.709} C_VEL
LIN {X 0,Y 235.408,Z 404.655,A -85,B 0,C 180,E1 -19626.859,E2 -19626.859} C_VEL
LIN {X 0,Y 235.255,Z 404.678,A -85,B 0,C 180,E1 -19630.326,E2 -19630.326} C_VEL
LIN {X 0,Y 235.116,Z 404.697,A -85,B 0,C 180,E1 -19635.606,E2 -19635.606} C_VEL
LIN {X 0,Y 235.022,Z 404.709,A -85,B 0,C 180,E1 -19639.205,E2 -19639.205} C_VEL
LIN {X 0,Y 234.983,Z 404.712,A -85,B 0,C 180,E1 -19642.881,E2 -19642.881} C_VEL
LIN {X 0,Y 234.971,Z 404.712,A -85,B 0,C 180,E1 -19646.657,E2 -19646.657} C_VEL
LIN {X 0,Y 234.934,Z 404.716,A -85,B 0,C 180,E1 -19650.568,E2 -19650.568} C_VEL
LIN {X 0,Y 234.962,Z 404.713,A -85,B 0,C 180,E1 -19654.633,E2 -19654.633} C_VEL
LIN {X 0,Y 234.943,Z 404.717,A -85,B 0,C 180,E1 -19658.945,E2 -19658.945} C_VEL
LIN {X 0,Y 234.889,Z 404.724,A -85,B 0,C 180,E1 -19663.486,E2 -19663.486} C_VEL
LIN {X 0,Y 234.881,Z 404.725,A -85,B 0,C 180,E1 -19666.513,E2 -19666.513} C_VEL
LIN {X 0,Y 234.92,Z 404.723,A -85,B 0,C 180,E1 -19671.079,E2 -19671.079} C_VEL
LIN {X 0,Y 235,Z 404.854,A -85,B 0,C 180,E1 -19673.546,E2 -19673.546} C_VEL
LIN {X 0,Y 235.464,Z 406.711,A -85,B 0,C 180,E1 -19674.501,E2 -19674.501} C_VEL
LIN {X 0,Y 244.565,Z 424.453,A -85,B 0,C 180,E1 -19676.633,E2 -19676.633} C_VEL
LIN {X 0,Y 251.701,Z 440.296,A -85,B 0,C 180,E1 -19678.227,E2 -19678.227} C_VEL
LIN {X 0,Y 255.022,Z 449.005,A -85,B 0,C 180,E1 -19678.973,E2 -19678.973} C_VEL
LIN {X 0,Y 253.073,Z 503.916,A -85,B 0,C 180,E1 -19680.479,E2 -19680.479} C_VEL
LIN {X 0,Y 252.344,Z 518.361,A -85,B 0,C 180,E1 -19680.984,E2 -19680.984} C_VEL
LIN {X 0,Y 251.084,Z 530.718,A -85,B 0,C 180,E1 -19681.7,E2 -19681.7} C_VEL
LIN {X 0,Y 249.511,Z 543.202,A -85,B 0,C 180,E1 -19682.76,E2 -19682.76} C_VEL
LIN {X 0,Y 247.502,Z 555.172,A -85,B 0,C 180,E1 -19684.114,E2 -19684.114} C_VEL
LIN {X 0,Y 245.351,Z 565.833,A -85,B 0,C 180,E1 -19685.684,E2 -19685.684} C_VEL
LIN {X 0,Y 243.2,Z 575.546,A -85,B 0,C 180,E1 -19687.487,E2 -19687.487} C_VEL
LIN {X 0,Y 241.129,Z 584.38,A -85,B 0,C 180,E1 -19689.528,E2 -19689.528} C_VEL
LIN {X 0,Y 238.823,Z 593,A -85,B 0,C 180,E1 -19692.002,E2 -19692.002} C_VEL
LIN {X 0,Y 236.884,Z 599.872,A -85,B 0,C 180,E1 -19694.513,E2 -19694.513} C_VEL
LIN {X 0,Y 235.376,Z 605.372,A -85,B 0,C 180,E1 -19697.06,E2 -19697.06} C_VEL
LIN {X 0,Y 234.242,Z 609.687,A -85,B 0,C 180,E1 -19699.629,E2 -19699.629} C_VEL
LIN {X 0,Y 233.716,Z 611.969,A -85,B 0,C 180,E1 -19701.353,E2 -19701.353} C_VEL
LIN {X 0,Y 233.094,Z 614.82,A -85,B 0,C 180,E1 -19704.26,E2 -19704.26} C_VEL
LIN {X 0,Y 232.9,Z 616.208,A -85,B 0,C 180,E1 -19706.54,E2 -19706.54} C_VEL
LIN {X 0,Y 232.802,Z 616.817,A -85,B 0,C 180,E1 -19708.27,E2 -19708.27} C_VEL
LIN {X 0,Y 232.768,Z 617.047,A -85,B 0,C 180,E1 -19710,E2 -19710} C_VEL
LIN {X 0,Y 232.802,Z 616.853,A -85,B 0,C 180,E1 -19711.73,E2 -19711.73} C_VEL
LIN {X 0,Y 232.899,Z 616.266,A -85,B 0,C 180,E1 -19713.46,E2 -19713.46} C_VEL
LIN {X 0,Y 233.3,Z 613.94,A -85,B 0,C 180,E1 -19716.921,E2 -19716.921} C_VEL
LIN {X 0,Y 233.989,Z 611.068,A -85,B 0,C 180,E1 -19719.509,E2 -19719.509} C_VEL
LIN {X 0,Y 234.946,Z 607.174,A -85,B 0,C 180,E1 -19722.087,E2 -19722.087} C_VEL
LIN {X 0,Y 236.299,Z 602.149,A -85,B 0,C 180,E1 -19724.644,E2 -19724.644} C_VEL
LIN {X 0,Y 238.035,Z 595.819,A -85,B 0,C 180,E1 -19727.173,E2 -19727.173} C_VEL
LIN {X 0,Y 240.265,Z 587.895,A -85,B 0,C 180,E1 -19729.657,E2 -19729.657} C_VEL
LIN {X 0,Y 242.462,Z 578.816,A -85,B 0,C 180,E1 -19731.943,E2 -19731.943} C_VEL
LIN {X 0,Y 244.686,Z 568.868,A -85,B 0,C 180,E1 -19733.936,E2 -19733.936} C_VEL
LIN {X 0,Y 247.109,Z 557.445,A -85,B 0,C 180,E1 -19735.705,E2 -19735.705} C_VEL
LIN {X 0,Y 249.118,Z 546.223,A -85,B 0,C 180,E1 -19737.06,E2 -19737.06} C_VEL
LIN {X 0,Y 250.75,Z 534.818,A -85,B 0,C 180,E1 -19738.114,E2 -19738.114} C_VEL
LIN {X 0,Y 252.086,Z 521.75,A -85,B 0,C 180,E1 -19738.974,E2 -19738.974} C_VEL
LIN {X 0,Y 252.948,Z 509.19,A -85,B 0,C 180,E1 -19739.493,E2 -19739.493} C_VEL
LIN {X 0,Y 253.691,Z 490.209,A -85,B 0,C 180,E1 -19740.015,E2 -19740.015} C_VEL
LIN {X 0,Y 255.123,Z 449.136,A -85,B 0,C 180,E1 -19741.144,E2 -19741.144} C_VEL
LIN {X 0,Y 248.838,Z 433.456,A -85,B 0,C 180,E1 -19742.553,E2 -19742.553} C_VEL
LIN {X 0,Y 241.01,Z 417.344,A -85,B 0,C 180,E1 -19744.324,E2 -19744.324} C_VEL
LIN {X 0,Y 236.78,Z 409.483,A -85,B 0,C 180,E1 -19745.316,E2 -19745.316} C_VEL
LIN {X 0,Y 235.428,Z 406.64,A -85,B 0,C 180,E1 -19745.667,E2 -19745.667} C_VEL
LIN {X 0,Y 234.97,Z 404.71,A -85,B 0,C 180,E1 -19746.742,E2 -19746.742} C_VEL
LIN {X 0,Y 234.887,Z 404.725,A -85,B 0,C 180,E1 -19751.168,E2 -19751.168} C_VEL
LIN {X 0,Y 234.905,Z 404.721,A -85,B 0,C 180,E1 -19755.894,E2 -19755.894} C_VEL
LIN {X 0,Y 234.909,Z 404.715,A -85,B 0,C 180,E1 -19758.837,E2 -19758.837} C_VEL
LIN {X 0,Y 234.958,Z 404.699,A -85,B 0,C 180,E1 -19761.086,E2 -19761.086} C_VEL
LIN {X 0,Y 234.964,Z 404.713,A -85,B 0,C 180,E1 -19765.367,E2 -19765.367} C_VEL
LIN {X 0,Y 234.973,Z 404.71,A -85,B 0,C 180,E1 -19770.157,E2 -19770.157} C_VEL
LIN {X 0,Y 234.998,Z 404.712,A -85,B 0,C 180,E1 -19773.794,E2 -19773.794} C_VEL
LIN {X 0,Y 235.032,Z 404.705,A -85,B 0,C 180,E1 -19778.972,E2 -19778.972} C_VEL
LIN {X 0,Y 235.101,Z 404.699,A -85,B 0,C 180,E1 -19783.059,E2 -19783.059} C_VEL
LIN {X 0,Y 235.151,Z 404.688,A -85,B 0,C 180,E1 -19787.924,E2 -19787.924} C_VEL
LIN {X 0,Y 235.395,Z 404.659,A -85,B 0,C 180,E1 -19791.415,E2 -19791.415} C_VEL
LIN {X 0,Y 235.411,Z 404.65,A -85,B 0,C 180,E1 -19793.141,E2 -19793.141} C_VEL
LIN {X 0,Y 235.601,Z 404.628,A -85,B 0,C 180,E1 -19798.291,E2 -19798.291} C_VEL
LIN {X 0,Y 235.6,Z 404.637,A -85,B 0,C 180,E1 -19801.709,E2 -19801.709} C_VEL
LIN {X 0,Y 235.373,Z 404.66,A -85,B 0,C 180,E1 -19806.86,E2 -19806.86} C_VEL
LIN {X 0,Y 235.218,Z 404.679,A -85,B 0,C 180,E1 -19810.327,E2 -19810.327} C_VEL
LIN {X 0,Y 235.118,Z 404.695,A -85,B 0,C 180,E1 -19815.606,E2 -19815.606} C_VEL
LIN {X 0,Y 235.013,Z 404.709,A -85,B 0,C 180,E1 -19819.205,E2 -19819.205} C_VEL
LIN {X 0,Y 234.991,Z 404.71,A -85,B 0,C 180,E1 -19820.527,E2 -19820.527} C_VEL
LIN {X 0,Y 234.353,Z 404.794,A -85,B 0,C 180,E1 -19821.958,E2 -19821.958} C_VEL
LIN {X 0,Y 231.483,Z 405.155,A -85,B 0,C 180,E1 -19824.291,E2 -19824.291} C_VEL
LIN {X 0,Y 229.016,Z 405.46,A -85,B 0,C 180,E1 -19826.194,E2 -19826.194} C_VEL
LIN {X 0,Y 227.95,Z 405.589,A -85,B 0,C 180,E1 -19827.672,E2 -19827.672} C_VEL
LIN {X 0,Y 227.86,Z 405.598,A -85,B 0,C 180,E1 -19828.174,E2 -19828.174} C_VEL
LIN {X 0,Y 227.87,Z 405.6,A -85,B 0,C 180,E1 -19831.622,E2 -19831.622} C_VEL
LIN {X 0,Y 227.883,Z 405.596,A -85,B 0,C 180,E1 -19835.871,E2 -19835.871} C_VEL
LIN {X 0,Y 227.829,Z 405.603,A -85,B 0,C 180,E1 -19840.376,E2 -19840.376} C_VEL
LIN {X 0,Y 227.838,Z 405.605,A -85,B 0,C 180,E1 -19845.192,E2 -19845.192} C_VEL
LIN {X 0,Y 227.862,Z 405.622,A -85,B 0,C 180,E1 -19848.552,E2 -19848.552} C_VEL
LIN {X 0,Y 229.918,Z 413.532,A -85,B 0,C 180,E1 -19852.632,E2 -19852.632} C_VEL
LIN {X 0,Y 230.414,Z 415.448,A -85,B 0,C 180,E1 -19853.489,E2 -19853.489} C_VEL
LIN {X 0,Y 232.476,Z 419.555,A -85,B 0,C 180,E1 -19854.015,E2 -19854.015} C_VEL
LIN {X 0,Y 238.821,Z 432.739,A -85,B 0,C 180,E1 -19855.579,E2 -19855.579} C_VEL
LIN {X 0,Y 244.701,Z 446.588,A -85,B 0,C 180,E1 -19856.987,E2 -19856.987} C_VEL
LIN {X 0,Y 246.021,Z 450.621,A -85,B 0,C 180,E1 -19857.323,E2 -19857.323} C_VEL
LIN {X 0,Y 248.456,Z 467.73,A -85,B 0,C 180,E1 -19858.251,E2 -19858.251} C_VEL
LIN {X 0,Y 246.219,Z 523.927,A -85,B 0,C 180,E1 -19859.854,E2 -19859.854} C_VEL
LIN {X 0,Y 244.965,Z 537.057,A -85,B 0,C 180,E1 -19860.514,E2 -19860.514} C_VEL
LIN {X 0,Y 243.389,Z 549.143,A -85,B 0,C 180,E1 -19861.428,E2 -19861.428} C_VEL
LIN {X 0,Y 241.24,Z 561.345,A -85,B 0,C 180,E1 -19862.687,E2 -19862.687} C_VEL
LIN {X 0,Y 238.84,Z 572.907,A -85,B 0,C 180,E1 -19864.276,E2 -19864.276} C_VEL
LIN {X 0,Y 236.349,Z 583.319,A -85,B 0,C 180,E1 -19866.099,E2 -19866.099} C_VEL
LIN {X 0,Y 234.181,Z 591.835,A -85,B 0,C 180,E1 -19867.967,E2 -19867.967} C_VEL
LIN {X 0,Y 232.227,Z 599.815,A -85,B 0,C 180,E1 -19870.132,E2 -19870.132} C_VEL
LIN {X 0,Y 230.129,Z 607.373,A -85,B 0,C 180,E1 -19872.677,E2 -19872.677} C_VEL
LIN {X 0,Y 228.019,Z 614.451,A -85,B 0,C 180,E1 -19875.725,E2 -19875.725} C_VEL
LIN {X 0,Y 226.913,Z 619.166,A -85,B 0,C 180,E1 -19878.385,E2 -19878.385} C_VEL
LIN {X 0,Y 226.151,Z 622.769,A -85,B 0,C 180,E1 -19881.061,E2 -19881.061} C_VEL
LIN {X 0,Y 225.823,Z 624.628,A -85,B 0,C 180,E1 -19882.848,E2 -19882.848} C_VEL
LIN {X 0,Y 225.577,Z 627.019,A -85,B 0,C 180,E1 -19886.427,E2 -19886.427} C_VEL
LIN {X 0,Y 225.618,Z 627.627,A -85,B 0,C 180,E1 -19888.215,E2 -19888.215} C_VEL
LIN {X 0,Y 225.674,Z 627.841,A -85,B 0,C 180,E1 -19890,E2 -19890} C_VEL
LIN {X 0,Y 225.618,Z 627.617,A -85,B 0,C 180,E1 -19891.785,E2 -19891.785} C_VEL
LIN {X 0,Y 225.584,Z 626.562,A -85,B 0,C 180,E1 -19894.474,E2 -19894.474} C_VEL
LIN {X 0,Y 225.823,Z 624.594,A -85,B 0,C 180,E1 -19897.151,E2 -19897.151} C_VEL
LIN {X 0,Y 226.357,Z 621.648,A -85,B 0,C 180,E1 -19899.832,E2 -19899.832} C_VEL
LIN {X 0,Y 227.257,Z 617.665,A -85,B 0,C 180,E1 -19902.502,E2 -19902.502} C_VEL
LIN {X 0,Y 228.571,Z 612.544,A -85,B 0,C 180,E1 -19905.15,E2 -19905.15} C_VEL
LIN {X 0,Y 230.395,Z 606.099,A -85,B 0,C 180,E1 -19907.76,E2 -19907.76} C_VEL
LIN {X 0,Y 232.489,Z 598.443,A -85,B 0,C 180,E1 -19910.226,E2 -19910.226} C_VEL
LIN {X 0,Y 234.62,Z 589.876,A -85,B 0,C 180,E1 -19912.453,E2 -19912.453} C_VEL
LIN {X 0,Y 237.141,Z 579.896,A -85,B 0,C 180,E1 -19914.513,E2 -19914.513} C_VEL
LIN {X 0,Y 239.694,Z 568.615,A -85,B 0,C 180,E1 -19916.326,E2 -19916.326} C_VEL
LIN {X 0,Y 241.817,Z 557.559,A -85,B 0,C 180,E1 -19917.711,E2 -19917.711} C_VEL
LIN {X 0,Y 243.779,Z 545.294,A -85,B 0,C 180,E1 -19918.874,E2 -19918.874} C_VEL
LIN {X 0,Y 245.466,Z 532.441,A -85,B 0,C 180,E1 -19919.709,E2 -19919.709} C_VEL
LIN {X 0,Y 246.465,Z 518.859,A -85,B 0,C 180,E1 -19920.276,E2 -19920.276} C_VEL
LIN {X 0,Y 248.256,Z 466.661,A -85,B 0,C 180,E1 -19921.765,E2 -19921.765} C_VEL
LIN {X 0,Y 245.685,Z 449.189,A -85,B 0,C 180,E1 -19922.726,E2 -19922.726} C_VEL
LIN {X 0,Y 239.445,Z 434.151,A -85,B 0,C 180,E1 -19924.215,E2 -19924.215} C_VEL
LIN {X 0,Y 233.938,Z 422.577,A -85,B 0,C 180,E1 -19925.557,E2 -19925.557} C_VEL
LIN {X 0,Y 230.412,Z 415.367,A -85,B 0,C 180,E1 -19926.454,E2 -19926.454} C_VEL
LIN {X 0,Y 228.41,Z 407.761,A -85,B 0,C 180,E1 -19930.252,E2 -19930.252} C_VEL
LIN {X 0,Y 227.842,Z 405.602,A -85,B 0,C 180,E1 -19931.453,E2 -19931.453} C_VEL
LIN {X 0,Y 227.836,Z 405.605,A -85,B 0,C 180,E1 -19935.192,E2 -19935.192} C_VEL
LIN {X 0,Y 227.827,Z 405.601,A -85,B 0,C 180,E1 -19939.623,E2 -19939.623} C_VEL
LIN {X 0,Y 227.882,Z 405.597,A -85,B 0,C 180,E1 -19944.128,E2 -19944.128} C_VEL
LIN {X 0,Y 227.867,Z 405.597,A -85,B 0,C 180,E1 -19948.377,E2 -19948.377} C_VEL
LIN {X 0,Y 227.88,Z 405.595,A -85,B 0,C 180,E1 -19952.444,E2 -19952.444} C_VEL
LIN {X 0,Y 227.926,Z 405.589,A -85,B 0,C 180,E1 -19956.369,E2 -19956.369} C_VEL
LIN {X 0,Y 227.956,Z 405.585,A -85,B 0,C 180,E1 -19960.176,E2 -19960.176} C_VEL
LIN {X 0,Y 228.059,Z 405.576,A -85,B 0,C 180,E1 -19963.898,E2 -19963.898} C_VEL
LIN {X 0,Y 228.075,Z 405.574,A -85,B 0,C 180,E1 -19967.543,E2 -19967.543} C_VEL
LIN {X 0,Y 228.265,Z 405.547,A -85,B 0,C 180,E1 -19971.144,E2 -19971.144} C_VEL
LIN {X 0,Y 228.32,Z 405.544,A -85,B 0,C 180,E1 -19972.928,E2 -19972.928} C_VEL
LIN {X 0,Y 228.556,Z 405.517,A -85,B 0,C 180,E1 -19978.238,E2 -19978.238} C_VEL
LIN {X 0,Y 228.558,Z 405.507,A -85,B 0,C 180,E1 -19981.762,E2 -19981.762} C_VEL
LIN {X 0,Y 228.36,Z 405.533,A -85,B 0,C 180,E1 -19987.071,E2 -19987.071} C_VEL
LIN {X 0,Y 228.173,Z 405.558,A -85,B 0,C 180,E1 -19990.65,E2 -19990.65} C_VEL
LIN {X 0,Y 228.059,Z 405.571,A -85,B 0,C 180,E1 -19996.102,E2 -19996.102} C_VEL
LIN {X 0,Y 227.957,Z 405.591,A -85,B 0,C 180,E1 -19999.824,E2 -19999.824} C_VEL
LIN {X 0,Y 227.926,Z 405.593,A -85,B 0,C 180,E1 -20003.631,E2 -20003.631} C_VEL
LIN {X 0,Y 227.888,Z 405.597,A -85,B 0,C 180,E1 -20007.555,E2 -20007.555} C_VEL
LIN {X 0,Y 227.875,Z 405.599,A -85,B 0,C 180,E1 -20011.622,E2 -20011.622} C_VEL
LIN {X 0,Y 227.903,Z 405.597,A -85,B 0,C 180,E1 -20015.868,E2 -20015.868} C_VEL
LIN {X 0,Y 227.838,Z 405.601,A -85,B 0,C 180,E1 -20020.374,E2 -20020.374} C_VEL
LIN {X 0,Y 227.831,Z 405.604,A -85,B 0,C 180,E1 -20025.194,E2 -20025.194} C_VEL
LIN {X 0,Y 227.826,Z 405.604,A -85,B 0,C 180,E1 -20029.623,E2 -20029.623} C_VEL
LIN {X 0,Y 227.902,Z 405.783,A -85,B 0,C 180,E1 -20032.584,E2 -20032.584} C_VEL
LIN {X 0,Y 228.225,Z 406.9,A -85,B 0,C 180,E1 -20033.192,E2 -20033.192} C_VEL
LIN {X 0,Y 230.353,Z 410.879,A -85,B 0,C 180,E1 -20033.741,E2 -20033.741} C_VEL
LIN {X 0,Y 237.388,Z 424.27,A -85,B 0,C 180,E1 -20035.47,E2 -20035.47} C_VEL
LIN {X 0,Y 244.793,Z 440.26,A -85,B 0,C 180,E1 -20037.212,E2 -20037.212} C_VEL
LIN {X 0,Y 248.968,Z 451.349,A -85,B 0,C 180,E1 -20038.203,E2 -20038.203} C_VEL
LIN {X 0,Y 246.949,Z 503.932,A -85,B 0,C 180,E1 -20039.665,E2 -20039.665} C_VEL
LIN {X 0,Y 246.23,Z 518.056,A -85,B 0,C 180,E1 -20040.164,E2 -20040.164} C_VEL
LIN {X 0,Y 244.876,Z 530.893,A -85,B 0,C 180,E1 -20040.915,E2 -20040.915} C_VEL
LIN {X 0,Y 243.212,Z 543.376,A -85,B 0,C 180,E1 -20041.994,E2 -20041.994} C_VEL
LIN {X 0,Y 241.155,Z 555.344,A -85,B 0,C 180,E1 -20043.38,E2 -20043.38} C_VEL
LIN {X 0,Y 238.906,Z 566.004,A -85,B 0,C 180,E1 -20044.984,E2 -20044.984} C_VEL
LIN {X 0,Y 236.658,Z 575.716,A -85,B 0,C 180,E1 -20046.829,E2 -20046.829} C_VEL
LIN {X 0,Y 234.499,Z 584.55,A -85,B 0,C 180,E1 -20048.922,E2 -20048.922} C_VEL
LIN {X 0,Y 232.083,Z 593.169,A -85,B 0,C 180,E1 -20051.46,E2 -20051.46} C_VEL
LIN {X 0,Y 230.033,Z 600.041,A -85,B 0,C 180,E1 -20054.04,E2 -20054.04} C_VEL
LIN {X 0,Y 228.459,Z 605.541,A -85,B 0,C 180,E1 -20056.661,E2 -20056.661} C_VEL
LIN {X 0,Y 227.259,Z 609.856,A -85,B 0,C 180,E1 -20059.307,E2 -20059.307} C_VEL
LIN {X 0,Y 226.691,Z 612.137,A -85,B 0,C 180,E1 -20061.083,E2 -20061.083} C_VEL
LIN {X 0,Y 225.966,Z 615.248,A -85,B 0,C 180,E1 -20064.426,E2 -20064.426} C_VEL
LIN {X 0,Y 225.808,Z 616.376,A -85,B 0,C 180,E1 -20066.431,E2 -20066.431} C_VEL
LIN {X 0,Y 225.721,Z 616.984,A -85,B 0,C 180,E1 -20068.216,E2 -20068.216} C_VEL
LIN {X 0,Y 225.684,Z 617.214,A -85,B 0,C 180,E1 -20070,E2 -20070} C_VEL
LIN {X 0,Y 225.72,Z 617.019,A -85,B 0,C 180,E1 -20071.785,E2 -20071.785} C_VEL
LIN {X 0,Y 225.808,Z 616.433,A -85,B 0,C 180,E1 -20073.569,E2 -20073.569} C_VEL
LIN {X 0,Y 226.036,Z 615.211,A -85,B 0,C 180,E1 -20075.755,E2 -20075.755} C_VEL
LIN {X 0,Y 226.717,Z 612.29,A -85,B 0,C 180,E1 -20078.917,E2 -20078.917} C_VEL
LIN {X 0,Y 227.595,Z 608.755,A -85,B 0,C 180,E1 -20081.579,E2 -20081.579} C_VEL
LIN {X 0,Y 228.897,Z 604.115,A -85,B 0,C 180,E1 -20084.22,E2 -20084.22} C_VEL
LIN {X 0,Y 230.9,Z 597.119,A -85,B 0,C 180,E1 -20087.264,E2 -20087.264} C_VEL
LIN {X 0,Y 233.182,Z 589.531,A -85,B 0,C 180,E1 -20089.821,E2 -20089.821} C_VEL
LIN {X 0,Y 235.38,Z 581,A -85,B 0,C 180,E1 -20092.113,E2 -20092.113} C_VEL
LIN {X 0,Y 237.714,Z 571.198,A -85,B 0,C 180,E1 -20094.219,E2 -20094.219} C_VEL
LIN {X 0,Y 240.181,Z 560.424,A -85,B 0,C 180,E1 -20096.035,E2 -20096.035} C_VEL
LIN {X 0,Y 242.235,Z 549.907,A -85,B 0,C 180,E1 -20097.425,E2 -20097.425} C_VEL
LIN {X 0,Y 244.2,Z 537.243,A -85,B 0,C 180,E1 -20098.703,E2 -20098.703} C_VEL
LIN {X 0,Y 245.67,Z 524.651,A -85,B 0,C 180,E1 -20099.621,E2 -20099.621} C_VEL
LIN {X 0,Y 246.727,Z 511.364,A -85,B 0,C 180,E1 -20100.233,E2 -20100.233} C_VEL
LIN {X 0,Y 248.737,Z 459.999,A -85,B 0,C 180,E1 -20101.68,E2 -20101.68} C_VEL
LIN {X 0,Y 248.889,Z 450.576,A -85,B 0,C 180,E1 -20101.973,E2 -20101.973} C_VEL
LIN {X 0,Y 242.562,Z 434.973,A -85,B 0,C 180,E1 -20103.457,E2 -20103.457} C_VEL
LIN {X 0,Y 234.512,Z 418.495,A -85,B 0,C 180,E1 -20105.379,E2 -20105.379} C_VEL
LIN {X 0,Y 229.619,Z 409.753,A -85,B 0,C 180,E1 -20106.589,E2 -20106.589} C_VEL
LIN {X 0,Y 228.17,Z 406.795,A -85,B 0,C 180,E1 -20107.008,E2 -20107.008} C_VEL
LIN {X 0,Y 227.886,Z 405.601,A -85,B 0,C 180,E1 -20107.704,E2 -20107.704} C_VEL
LIN {X 0,Y 227.816,Z 405.606,A -85,B 0,C 180,E1 -20112.742,E2 -20112.742} C_VEL
LIN {X 0,Y 227.842,Z 405.604,A -85,B 0,C 180,E1 -20117.265,E2 -20117.265} C_VEL
LIN {X 0,Y 227.874,Z 405.587,A -85,B 0,C 180,E1 -20121.915,E2 -20121.915} C_VEL
LIN {X 0,Y 227.894,Z 405.592,A -85,B 0,C 180,E1 -20126.373,E2 -20126.373} C_VEL
LIN {X 0,Y 227.923,Z 405.588,A -85,B 0,C 180,E1 -20130.438,E2 -20130.438} C_VEL
LIN {X 0,Y 227.933,Z 405.585,A -85,B 0,C 180,E1 -20134.426,E2 -20134.426} C_VEL
LIN {X 0,Y 227.996,Z 405.585,A -85,B 0,C 180,E1 -20138.29,E2 -20138.29} C_VEL
LIN {X 0,Y 228.04,Z 405.579,A -85,B 0,C 180,E1 -20142.825,E2 -20142.825} C_VEL
LIN {X 0,Y 228.098,Z 405.564,A -85,B 0,C 180,E1 -20147.545,E2 -20147.545} C_VEL
LIN {X 0,Y 228.33,Z 405.54,A -85,B 0,C 180,E1 -20151.147,E2 -20151.147} C_VEL
LIN {X 0,Y 228.363,Z 405.527,A -85,B 0,C 180,E1 -20152.929,E2 -20152.929} C_VEL
LIN {X 0,Y 228.559,Z 405.505,A -85,B 0,C 180,E1 -20158.238,E2 -20158.238} C_VEL
LIN {X 0,Y 228.559,Z 405.515,A -85,B 0,C 180,E1 -20161.762,E2 -20161.762} C_VEL
LIN {X 0,Y 228.323,Z 405.539,A -85,B 0,C 180,E1 -20167.072,E2 -20167.072} C_VEL
LIN {X 0,Y 228.15,Z 405.559,A -85,B 0,C 180,E1 -20170.651,E2 -20170.651} C_VEL
LIN {X 0,Y 228.07,Z 405.575,A -85,B 0,C 180,E1 -20174.272,E2 -20174.272} C_VEL
LIN {X 0,Y 228.007,Z 405.577,A -85,B 0,C 180,E1 -20177.953,E2 -20177.953} C_VEL
LIN {X 0,Y 227.934,Z 405.583,A -85,B 0,C 180,E1 -20182.329,E2 -20182.329} C_VEL
LIN {X 0,Y 227.945,Z 405.59,A -85,B 0,C 180,E1 -20186.602,E2 -20186.602} C_VEL
LIN {X 0,Y 227.86,Z 405.598,A -85,B 0,C 180,E1 -20188.174,E2 -20188.174} C_VEL
LIN {X 0,Y 227.179,Z 405.686,A -85,B 0,C 180,E1 -20189.649,E2 -20189.649} C_VEL
LIN {X 0,Y 224.306,Z 406.042,A -85,B 0,C 180,E1 -20192.057,E2 -20192.057} C_VEL
LIN {X 0,Y 221.878,Z 406.344,A -85,B 0,C 180,E1 -20194.021,E2 -20194.021} C_VEL
LIN {X 0,Y 220.85,Z 406.474,A -85,B 0,C 180,E1 -20195.547,E2 -20195.547} C_VEL
LIN {X 0,Y 220.772,Z 406.478,A -85,B 0,C 180,E1 -20196.064,E2 -20196.064} C_VEL
LIN {X 0,Y 220.798,Z 406.479,A -85,B 0,C 180,E1 -20200.188,E2 -20200.188} C_VEL
LIN {X 0,Y 220.778,Z 406.485,A -85,B 0,C 180,E1 -20204.453,E2 -20204.453} C_VEL
LIN {X 0,Y 220.789,Z 406.544,A -85,B 0,C 180,E1 -20207.48,E2 -20207.48} C_VEL
LIN {X 0,Y 223.026,Z 414.994,A -85,B 0,C 180,E1 -20212.05,E2 -20212.05} C_VEL
LIN {X 0,Y 225.205,Z 419.254,A -85,B 0,C 180,E1 -20212.656,E2 -20212.656} C_VEL
LIN {X 0,Y 232.318,Z 433.607,A -85,B 0,C 180,E1 -20214.511,E2 -20214.511} C_VEL
LIN {X 0,Y 238.501,Z 447.936,A -85,B 0,C 180,E1 -20216.067,E2 -20216.067} C_VEL
LIN {X 0,Y 240.191,Z 452.669,A -85,B 0,C 180,E1 -20216.503,E2 -20216.503} C_VEL
LIN {X 0,Y 242.41,Z 468.8,A -85,B 0,C 180,E1 -20217.404,E2 -20217.404} C_VEL
LIN {X 0,Y 240.073,Z 524.206,A -85,B 0,C 180,E1 -20219.022,E2 -20219.022} C_VEL
LIN {X 0,Y 238.68,Z 537.722,A -85,B 0,C 180,E1 -20219.723,E2 -20219.723} C_VEL
LIN {X 0,Y 237.014,Z 550.092,A -85,B 0,C 180,E1 -20220.707,E2 -20220.707} C_VEL
LIN {X 0,Y 234.953,Z 561.182,A -85,B 0,C 180,E1 -20221.892,E2 -20221.892} C_VEL
LIN {X 0,Y 232.464,Z 572.744,A -85,B 0,C 180,E1 -20223.516,E2 -20223.516} C_VEL
LIN {X 0,Y 229.879,Z 583.156,A -85,B 0,C 180,E1 -20225.382,E2 -20225.382} C_VEL
LIN {X 0,Y 227.576,Z 591.669,A -85,B 0,C 180,E1 -20227.292,E2 -20227.292} C_VEL
LIN {X 0,Y 225.693,Z 598.937,A -85,B 0,C 180,E1 -20229.302,E2 -20229.302} C_VEL
LIN {X 0,Y 223.62,Z 606.05,A -85,B 0,C 180,E1 -20231.682,E2 -20231.682} C_VEL
LIN {X 0,Y 221.722,Z 612.467,A -85,B 0,C 180,E1 -20234.369,E2 -20234.369} C_VEL
LIN {X 0,Y 220.281,Z 617.566,A -85,B 0,C 180,E1 -20237.095,E2 -20237.095} C_VEL
LIN {X 0,Y 219.341,Z 621.53,A -85,B 0,C 180,E1 -20239.849,E2 -20239.849} C_VEL
LIN {X 0,Y 218.762,Z 624.461,A -85,B 0,C 180,E1 -20242.616,E2 -20242.616} C_VEL
LIN {X 0,Y 218.481,Z 626.586,A -85,B 0,C 180,E1 -20245.708,E2 -20245.708} C_VEL
LIN {X 0,Y 218.517,Z 627.46,A -85,B 0,C 180,E1 -20248.157,E2 -20248.157} C_VEL
LIN {X 0,Y 218.59,Z 627.674,A -85,B 0,C 180,E1 -20250,E2 -20250} C_VEL
LIN {X 0,Y 218.518,Z 627.449,A -85,B 0,C 180,E1 -20251.843,E2 -20251.843} C_VEL
LIN {X 0,Y 218.481,Z 626.569,A -85,B 0,C 180,E1 -20254.291,E2 -20254.291} C_VEL
LIN {X 0,Y 218.761,Z 624.426,A -85,B 0,C 180,E1 -20257.383,E2 -20257.383} C_VEL
LIN {X 0,Y 219.34,Z 621.479,A -85,B 0,C 180,E1 -20260.15,E2 -20260.15} C_VEL
LIN {X 0,Y 220.276,Z 617.495,A -85,B 0,C 180,E1 -20262.905,E2 -20262.905} C_VEL
LIN {X 0,Y 222.021,Z 611.375,A -85,B 0,C 180,E1 -20266.08,E2 -20266.08} C_VEL
LIN {X 0,Y 223.95,Z 604.693,A -85,B 0,C 180,E1 -20268.763,E2 -20268.763} C_VEL
LIN {X 0,Y 226.104,Z 596.926,A -85,B 0,C 180,E1 -20271.254,E2 -20271.254} C_VEL
LIN {X 0,Y 228.556,Z 587.903,A -85,B 0,C 180,E1 -20273.562,E2 -20273.562} C_VEL
LIN {X 0,Y 231.258,Z 577.404,A -85,B 0,C 180,E1 -20275.662,E2 -20275.662} C_VEL
LIN {X 0,Y 233.966,Z 565.585,A -85,B 0,C 180,E1 -20277.506,E2 -20277.506} C_VEL
LIN {X 0,Y 236.289,Z 553.676,A -85,B 0,C 180,E1 -20278.903,E2 -20278.903} C_VEL
LIN {X 0,Y 237.999,Z 542.578,A -85,B 0,C 180,E1 -20279.888,E2 -20279.888} C_VEL
LIN {X 0,Y 239.67,Z 529.042,A -85,B 0,C 180,E1 -20280.717,E2 -20280.717} C_VEL
LIN {X 0,Y 240.497,Z 514.997,A -85,B 0,C 180,E1 -20281.243,E2 -20281.243} C_VEL
LIN {X 0,Y 242.23,Z 467.806,A -85,B 0,C 180,E1 -20282.606,E2 -20282.606} C_VEL
LIN {X 0,Y 239.931,Z 451.77,A -85,B 0,C 180,E1 -20283.516,E2 -20283.516} C_VEL
LIN {X 0,Y 234.125,Z 437.623,A -85,B 0,C 180,E1 -20284.972,E2 -20284.972} C_VEL
LIN {X 0,Y 227.413,Z 423.555,A -85,B 0,C 180,E1 -20286.695,E2 -20286.695} C_VEL
LIN {X 0,Y 223.045,Z 414.981,A -85,B 0,C 180,E1 -20287.888,E2 -20287.888} C_VEL
LIN {X 0,Y 220.781,Z 406.483,A -85,B 0,C 180,E1 -20292.506,E2 -20292.506} C_VEL
LIN {X 0,Y 220.768,Z 406.481,A -85,B 0,C 180,E1 -20297.07,E2 -20297.07} C_VEL
LIN {X 0,Y 220.807,Z 406.478,A -85,B 0,C 180,E1 -20300.463,E2 -20300.463} C_VEL
LIN {X 0,Y 220.802,Z 406.475,A -85,B 0,C 180,E1 -20305.045,E2 -20305.045} C_VEL
LIN {X 0,Y 220.834,Z 406.474,A -85,B 0,C 180,E1 -20309.39,E2 -20309.39} C_VEL
LIN {X 0,Y 220.895,Z 406.468,A -85,B 0,C 180,E1 -20313.55,E2 -20313.55} C_VEL
LIN {X 0,Y 220.925,Z 406.464,A -85,B 0,C 180,E1 -20317.559,E2 -20317.559} C_VEL
LIN {X 0,Y 220.986,Z 406.459,A -85,B 0,C 180,E1 -20322.57,E2 -20322.57} C_VEL
LIN {X 0,Y 221.014,Z 406.454,A -85,B 0,C 180,E1 -20327.139,E2 -20327.139} C_VEL
LIN {X 0,Y 221.203,Z 406.425,A -85,B 0,C 180,E1 -20330.859,E2 -20330.859} C_VEL
LIN {X 0,Y 221.139,Z 406.433,A -85,B 0,C 180,E1 -20334.529,E2 -20334.529} C_VEL
LIN {X 0,Y 221.514,Z 406.394,A -85,B 0,C 180,E1 -20338.182,E2 -20338.182} C_VEL
LIN {X 0,Y 221.516,Z 406.384,A -85,B 0,C 180,E1 -20341.818,E2 -20341.818} C_VEL
LIN {X 0,Y 221.313,Z 406.411,A -85,B 0,C 180,E1 -20347.298,E2 -20347.298} C_VEL
LIN {X 0,Y 221.118,Z 406.436,A -85,B 0,C 180,E1 -20350.994,E2 -20350.994} C_VEL
LIN {X 0,Y 221.019,Z 406.445,A -85,B 0,C 180,E1 -20356.63,E2 -20356.63} C_VEL
LIN {X 0,Y 220.912,Z 406.464,A -85,B 0,C 180,E1 -20360.484,E2 -20360.484} C_VEL
LIN {X 0,Y 220.874,Z 406.471,A -85,B 0,C 180,E1 -20364.434,E2 -20364.434} C_VEL
LIN {X 0,Y 220.838,Z 406.476,A -85,B 0,C 180,E1 -20368.514,E2 -20368.514} C_VEL
LIN {X 0,Y 220.826,Z 406.477,A -85,B 0,C 180,E1 -20372.755,E2 -20372.755} C_VEL
LIN {X 0,Y 220.839,Z 406.472,A -85,B 0,C 180,E1 -20377.288,E2 -20377.288} C_VEL
LIN {X 0,Y 220.78,Z 406.482,A -85,B 0,C 180,E1 -20381.951,E2 -20381.951} C_VEL
LIN {X 0,Y 220.771,Z 406.486,A -85,B 0,C 180,E1 -20385.545,E2 -20385.545} C_VEL
LIN {X 0,Y 220.808,Z 406.481,A -85,B 0,C 180,E1 -20390.463,E2 -20390.463} C_VEL
LIN {X 0,Y 220.828,Z 406.61,A -85,B 0,C 180,E1 -20391.495,E2 -20391.495} C_VEL
LIN {X 0,Y 220.929,Z 407.173,A -85,B 0,C 180,E1 -20391.764,E2 -20391.764} C_VEL
LIN {X 0,Y 222.278,Z 409.986,A -85,B 0,C 180,E1 -20392.152,E2 -20392.152} C_VEL
LIN {X 0,Y 223.966,Z 412.506,A -85,B 0,C 180,E1 -20392.59,E2 -20392.59} C_VEL
LIN {X 0,Y 231.413,Z 426.339,A -85,B 0,C 180,E1 -20394.516,E2 -20394.516} C_VEL
LIN {X 0,Y 239.32,Z 443.51,A -85,B 0,C 180,E1 -20396.472,E2 -20396.472} C_VEL
LIN {X 0,Y 242.867,Z 452.662,A -85,B 0,C 180,E1 -20397.345,E2 -20397.345} C_VEL
LIN {X 0,Y 240.862,Z 504.005,A -85,B 0,C 180,E1 -20398.81,E2 -20398.81} C_VEL
LIN {X 0,Y 240.064,Z 518.736,A -85,B 0,C 180,E1 -20399.346,E2 -20399.346} C_VEL
LIN {X 0,Y 238.713,Z 531.068,A -85,B 0,C 180,E1 -20400.089,E2 -20400.089} C_VEL
LIN {X 0,Y 236.96,Z 543.55,A -85,B 0,C 180,E1 -20401.187,E2 -20401.187} C_VEL
LIN {X 0,Y 234.843,Z 555.516,A -85,B 0,C 180,E1 -20402.605,E2 -20402.605} C_VEL
LIN {X 0,Y 232.488,Z 566.175,A -85,B 0,C 180,E1 -20404.244,E2 -20404.244} C_VEL
LIN {X 0,Y 230.143,Z 575.886,A -85,B 0,C 180,E1 -20406.133,E2 -20406.133} C_VEL
LIN {X 0,Y 227.894,Z 584.72,A -85,B 0,C 180,E1 -20408.28,E2 -20408.28} C_VEL
LIN {X 0,Y 225.365,Z 593.338,A -85,B 0,C 180,E1 -20410.887,E2 -20410.887} C_VEL
LIN {X 0,Y 223.197,Z 600.211,A -85,B 0,C 180,E1 -20413.538,E2 -20413.538} C_VEL
LIN {X 0,Y 221.561,Z 605.709,A -85,B 0,C 180,E1 -20416.237,E2 -20416.237} C_VEL
LIN {X 0,Y 220.267,Z 610.024,A -85,B 0,C 180,E1 -20418.963,E2 -20418.963} C_VEL
LIN {X 0,Y 219.658,Z 612.306,A -85,B 0,C 180,E1 -20420.795,E2 -20420.795} C_VEL
LIN {X 0,Y 219.207,Z 614.16,A -85,B 0,C 180,E1 -20422.632,E2 -20422.632} C_VEL
LIN {X 0,Y 218.887,Z 615.553,A -85,B 0,C 180,E1 -20424.473,E2 -20424.473} C_VEL
LIN {X 0,Y 218.721,Z 616.543,A -85,B 0,C 180,E1 -20426.316,E2 -20426.316} C_VEL
LIN {X 0,Y 218.641,Z 617.151,A -85,B 0,C 180,E1 -20428.158,E2 -20428.158} C_VEL
LIN {X 0,Y 218.602,Z 617.38,A -85,B 0,C 180,E1 -20430,E2 -20430} C_VEL
LIN {X 0,Y 218.641,Z 617.186,A -85,B 0,C 180,E1 -20431.842,E2 -20431.842} C_VEL
LIN {X 0,Y 218.721,Z 616.6,A -85,B 0,C 180,E1 -20433.685,E2 -20433.685} C_VEL
LIN {X 0,Y 219.209,Z 614.273,A -85,B 0,C 180,E1 -20437.368,E2 -20437.368} C_VEL
LIN {X 0,Y 219.966,Z 611.401,A -85,B 0,C 180,E1 -20440.121,E2 -20440.121} C_VEL
LIN {X 0,Y 221.044,Z 607.507,A -85,B 0,C 180,E1 -20442.86,E2 -20442.86} C_VEL
LIN {X 0,Y 222.545,Z 602.481,A -85,B 0,C 180,E1 -20445.571,E2 -20445.571} C_VEL
LIN {X 0,Y 224.53,Z 596.148,A -85,B 0,C 180,E1 -20448.241,E2 -20448.241} C_VEL
LIN {X 0,Y 226.95,Z 588.224,A -85,B 0,C 180,E1 -20450.863,E2 -20450.863} C_VEL
LIN {X 0,Y 229.033,Z 580.307,A -85,B 0,C 180,E1 -20452.99,E2 -20452.99} C_VEL
LIN {X 0,Y 231.516,Z 570.295,A -85,B 0,C 180,E1 -20455.151,E2 -20455.151} C_VEL
LIN {X 0,Y 234.13,Z 559.191,A -85,B 0,C 180,E1 -20457.002,E2 -20457.002} C_VEL
LIN {X 0,Y 236.273,Z 548.307,A -85,B 0,C 180,E1 -20458.42,E2 -20458.42} C_VEL
LIN {X 0,Y 238.175,Z 536.274,A -85,B 0,C 180,E1 -20459.621,E2 -20459.621} C_VEL
LIN {X 0,Y 239.684,Z 523.461,A -85,B 0,C 180,E1 -20460.536,E2 -20460.536} C_VEL
LIN {X 0,Y 240.717,Z 509.729,A -85,B 0,C 180,E1 -20461.143,E2 -20461.143} C_VEL
LIN {X 0,Y 242.976,Z 452.799,A -85,B 0,C 180,E1 -20462.775,E2 -20462.775} C_VEL
LIN {X 0,Y 237.316,Z 438.784,A -85,B 0,C 180,E1 -20464.166,E2 -20464.166} C_VEL
LIN {X 0,Y 229.608,Z 422.74,A -85,B 0,C 180,E1 -20466.096,E2 -20466.096} C_VEL
LIN {X 0,Y 222.996,Z 410.848,A -85,B 0,C 180,E1 -20467.826,E2 -20467.826} C_VEL
LIN {X 0,Y 221.163,Z 407.992,A -85,B 0,C 180,E1 -20468.313,E2 -20468.313} C_VEL
LIN {X 0,Y 220.887,Z 406.993,A -85,B 0,C 180,E1 -20468.449,E2 -20468.449} C_VEL
LIN {X 0,Y 220.794,Z 406.481,A -85,B 0,C 180,E1 -20468.941,E2 -20468.941} C_VEL
LIN {X 0,Y 220.771,Z 406.482,A -85,B 0,C 180,E1 -20472.93,E2 -20472.93} C_VEL
LIN {X 0,Y 220.793,Z 406.483,A -85,B 0,C 180,E1 -20477.064,E2 -20477.064} C_VEL
LIN {X 0,Y 220.815,Z 406.457,A -85,B 0,C 180,E1 -20480.464,E2 -20480.464} C_VEL
LIN {X 0,Y 220.838,Z 406.471,A -85,B 0,C 180,E1 -20482.795,E2 -20482.795} C_VEL
LIN {X 0,Y 220.828,Z 406.476,A -85,B 0,C 180,E1 -20487.246,E2 -20487.246} C_VEL
LIN {X 0,Y 220.841,Z 406.472,A -85,B 0,C 180,E1 -20491.487,E2 -20491.487} C_VEL
LIN {X 0,Y 220.877,Z 406.461,A -85,B 0,C 180,E1 -20495.566,E2 -20495.566} C_VEL
LIN {X 0,Y 220.914,Z 406.462,A -85,B 0,C 180,E1 -20499.516,E2 -20499.516} C_VEL
LIN {X 0,Y 221.021,Z 406.453,A -85,B 0,C 180,E1 -20503.37,E2 -20503.37} C_VEL
LIN {X 0,Y 221.121,Z 406.44,A -85,B 0,C 180,E1 -20509.006,E2 -20509.006} C_VEL
LIN {X 0,Y 221.3,Z 406.406,A -85,B 0,C 180,E1 -20512.702,E2 -20512.702} C_VEL
LIN {X 0,Y 221.517,Z 406.382,A -85,B 0,C 180,E1 -20518.182,E2 -20518.182} C_VEL
LIN {X 0,Y 221.517,Z 406.392,A -85,B 0,C 180,E1 -20521.818,E2 -20521.818} C_VEL
LIN {X 0,Y 221.259,Z 406.42,A -85,B 0,C 180,E1 -20527.299,E2 -20527.299} C_VEL
LIN {X 0,Y 221.071,Z 406.438,A -85,B 0,C 180,E1 -20530.996,E2 -20530.996} C_VEL
LIN {X 0,Y 221.001,Z 406.455,A -85,B 0,C 180,E1 -20534.738,E2 -20534.738} C_VEL
LIN {X 0,Y 220.926,Z 406.462,A -85,B 0,C 180,E1 -20538.549,E2 -20538.549} C_VEL
LIN {X 0,Y 220.9,Z 406.459,A -85,B 0,C 180,E1 -20542.683,E2 -20542.683} C_VEL
LIN {X 0,Y 220.887,Z 406.47,A -85,B 0,C 180,E1 -20547.014,E2 -20547.014} C_VEL
LIN {X 0,Y 220.841,Z 406.473,A -85,B 0,C 180,E1 -20550.767,E2 -20550.767} C_VEL
LIN {X 0,Y 220.804,Z 406.478,A -85,B 0,C 180,E1 -20554.955,E2 -20554.955} C_VEL
LIN {X 0,Y 220.772,Z 406.478,A -85,B 0,C 180,E1 -20556.064,E2 -20556.064} C_VEL
LIN {X 0,Y 220.114,Z 406.565,A -85,B 0,C 180,E1 -20557.587,E2 -20557.587} C_VEL
LIN {X 0,Y 217.245,Z 406.923,A -85,B 0,C 180,E1 -20560.072,E2 -20560.072} C_VEL
LIN {X 0,Y 214.809,Z 407.227,A -85,B 0,C 180,E1 -20562.101,E2 -20562.101} C_VEL
LIN {X 0,Y 213.784,Z 407.355,A -85,B 0,C 180,E1 -20563.679,E2 -20563.679} C_VEL
LIN {X 0,Y 213.711,Z 407.363,A -85,B 0,C 180,E1 -20564.213,E2 -20564.213} C_VEL
LIN {X 0,Y 213.75,Z 407.473,A -85,B 0,C 180,E1 -20566.332,E2 -20566.332} C_VEL
LIN {X 0,Y 215.677,Z 414.808,A -85,B 0,C 180,E1 -20570.522,E2 -20570.522} C_VEL
LIN {X 0,Y 218.145,Z 419.341,A -85,B 0,C 180,E1 -20571.238,E2 -20571.238} C_VEL
LIN {X 0,Y 225.165,Z 433.072,A -85,B 0,C 180,E1 -20573.188,E2 -20573.188} C_VEL
LIN {X 0,Y 232.091,Z 448.709,A -85,B 0,C 180,E1 -20575.03,E2 -20575.03} C_VEL
LIN {X 0,Y 234.466,Z 455.217,A -85,B 0,C 180,E1 -20575.67,E2 -20575.67} C_VEL
LIN {X 0,Y 236.41,Z 469.187,A -85,B 0,C 180,E1 -20576.488,E2 -20576.488} C_VEL
LIN {X 0,Y 234.047,Z 523.721,A -85,B 0,C 180,E1 -20578.114,E2 -20578.114} C_VEL
LIN {X 0,Y 232.705,Z 536.949,A -85,B 0,C 180,E1 -20578.809,E2 -20578.809} C_VEL
LIN {X 0,Y 230.852,Z 549.932,A -85,B 0,C 180,E1 -20579.846,E2 -20579.846} C_VEL
LIN {X 0,Y 228.714,Z 561.02,A -85,B 0,C 180,E1 -20581.054,E2 -20581.054} C_VEL
LIN {X 0,Y 226.117,Z 572.58,A -85,B 0,C 180,E1 -20582.712,E2 -20582.712} C_VEL
LIN {X 0,Y 223.424,Z 582.991,A -85,B 0,C 180,E1 -20584.622,E2 -20584.622} C_VEL
LIN {X 0,Y 221.033,Z 591.505,A -85,B 0,C 180,E1 -20586.581,E2 -20586.581} C_VEL
LIN {X 0,Y 218.858,Z 599.409,A -85,B 0,C 180,E1 -20588.837,E2 -20588.837} C_VEL
LIN {X 0,Y 216.527,Z 607.039,A -85,B 0,C 180,E1 -20591.55,E2 -20591.55} C_VEL
LIN {X 0,Y 214.251,Z 614.119,A -85,B 0,C 180,E1 -20594.786,E2 -20594.786} C_VEL
LIN {X 0,Y 212.956,Z 618.833,A -85,B 0,C 180,E1 -20597.613,E2 -20597.613} C_VEL
LIN {X 0,Y 212.076,Z 622.435,A -85,B 0,C 180,E1 -20600.462,E2 -20600.462} C_VEL
LIN {X 0,Y 211.69,Z 624.293,A -85,B 0,C 180,E1 -20602.368,E2 -20602.368} C_VEL
LIN {X 0,Y 211.394,Z 626.543,A -85,B 0,C 180,E1 -20605.855,E2 -20605.855} C_VEL
LIN {X 0,Y 211.42,Z 627.293,A -85,B 0,C 180,E1 -20608.095,E2 -20608.095} C_VEL
LIN {X 0,Y 211.49,Z 627.507,A -85,B 0,C 180,E1 -20610,E2 -20610} C_VEL
LIN {X 0,Y 211.421,Z 627.282,A -85,B 0,C 180,E1 -20611.905,E2 -20611.905} C_VEL
LIN {X 0,Y 211.393,Z 626.525,A -85,B 0,C 180,E1 -20614.145,E2 -20614.145} C_VEL
LIN {X 0,Y 211.69,Z 624.257,A -85,B 0,C 180,E1 -20617.631,E2 -20617.631} C_VEL
LIN {X 0,Y 212.342,Z 621.311,A -85,B 0,C 180,E1 -20620.488,E2 -20620.488} C_VEL
LIN {X 0,Y 213.31,Z 617.326,A -85,B 0,C 180,E1 -20623.334,E2 -20623.334} C_VEL
LIN {X 0,Y 215.165,Z 611.205,A -85,B 0,C 180,E1 -20626.607,E2 -20626.607} C_VEL
LIN {X 0,Y 217.223,Z 604.523,A -85,B 0,C 180,E1 -20629.367,E2 -20629.367} C_VEL
LIN {X 0,Y 219.391,Z 597.069,A -85,B 0,C 180,E1 -20631.833,E2 -20631.833} C_VEL
LIN {X 0,Y 222.042,Z 587.732,A -85,B 0,C 180,E1 -20634.297,E2 -20634.297} C_VEL
LIN {X 0,Y 224.845,Z 577.232,A -85,B 0,C 180,E1 -20636.45,E2 -20636.45} C_VEL
LIN {X 0,Y 227.702,Z 565.414,A -85,B 0,C 180,E1 -20638.33,E2 -20638.33} C_VEL
LIN {X 0,Y 230.112,Z 553.503,A -85,B 0,C 180,E1 -20639.755,E2 -20639.755} C_VEL
LIN {X 0,Y 231.881,Z 542.404,A -85,B 0,C 180,E1 -20640.761,E2 -20640.761} C_VEL
LIN {X 0,Y 233.56,Z 529.312,A -85,B 0,C 180,E1 -20641.581,E2 -20641.581} C_VEL
LIN {X 0,Y 234.403,Z 516.371,A -85,B 0,C 180,E1 -20642.096,E2 -20642.096} C_VEL
LIN {X 0,Y 236.186,Z 468.388,A -85,B 0,C 180,E1 -20643.521,E2 -20643.521} C_VEL
LIN {X 0,Y 234.146,Z 454.122,A -85,B 0,C 180,E1 -20644.367,E2 -20644.367} C_VEL
LIN {X 0,Y 227.702,Z 438.51,A -85,B 0,C 180,E1 -20646.068,E2 -20646.068} C_VEL
LIN {X 0,Y 220.45,Z 423.621,A -85,B 0,C 180,E1 -20648.043,E2 -20648.043} C_VEL
LIN {X 0,Y 215.664,Z 414.667,A -85,B 0,C 180,E1 -20649.474,E2 -20649.474} C_VEL
LIN {X 0,Y 213.708,Z 407.361,A -85,B 0,C 180,E1 -20653.678,E2 -20653.678} C_VEL
LIN {X 0,Y 213.708,Z 407.36,A -85,B 0,C 180,E1 -20656.343,E2 -20656.343} C_VEL
LIN {X 0,Y 213.718,Z 407.357,A -85,B 0,C 180,E1 -20659.143,E2 -20659.143} C_VEL
LIN {X 0,Y 213.744,Z 407.358,A -85,B 0,C 180,E1 -20663.712,E2 -20663.712} C_VEL
LIN {X 0,Y 213.768,Z 407.353,A -85,B 0,C 180,E1 -20668.262,E2 -20668.262} C_VEL
LIN {X 0,Y 213.827,Z 407.345,A -85,B 0,C 180,E1 -20672.603,E2 -20672.603} C_VEL
LIN {X 0,Y 213.863,Z 407.341,A -85,B 0,C 180,E1 -20676.946,E2 -20676.946} C_VEL
LIN {X 0,Y 213.935,Z 407.335,A -85,B 0,C 180,E1 -20682.304,E2 -20682.304} C_VEL
LIN {X 0,Y 213.955,Z 407.332,A -85,B 0,C 180,E1 -20686.707,E2 -20686.707} C_VEL
LIN {X 0,Y 214.141,Z 407.303,A -85,B 0,C 180,E1 -20690.555,E2 -20690.555} C_VEL
LIN {X 0,Y 214.1,Z 407.311,A -85,B 0,C 180,E1 -20694.349,E2 -20694.349} C_VEL
LIN {X 0,Y 214.447,Z 407.273,A -85,B 0,C 180,E1 -20698.122,E2 -20698.122} C_VEL
LIN {X 0,Y 214.552,Z 407.254,A -85,B 0,C 180,E1 -20700,E2 -20700} C_VEL
LIN {X 0,Y 214.449,Z 407.264,A -85,B 0,C 180,E1 -20701.878,E2 -20701.878} C_VEL
LIN {X 0,Y 214.25,Z 407.291,A -85,B 0,C 180,E1 -20707.54,E2 -20707.54} C_VEL
LIN {X 0,Y 214.049,Z 407.315,A -85,B 0,C 180,E1 -20711.362,E2 -20711.362} C_VEL
LIN {X 0,Y 213.936,Z 407.335,A -85,B 0,C 180,E1 -20715.237,E2 -20715.237} C_VEL
LIN {X 0,Y 213.878,Z 407.343,A -85,B 0,C 180,E1 -20719.184,E2 -20719.184} C_VEL
LIN {X 0,Y 213.857,Z 407.344,A -85,B 0,C 180,E1 -20723.226,E2 -20723.226} C_VEL
LIN {X 0,Y 213.83,Z 407.347,A -85,B 0,C 180,E1 -20727.45,E2 -20727.45} C_VEL
LIN {X 0,Y 213.781,Z 407.355,A -85,B 0,C 180,E1 -20731.736,E2 -20731.736} C_VEL
LIN {X 0,Y 213.755,Z 407.357,A -85,B 0,C 180,E1 -20736.286,E2 -20736.286} C_VEL
LIN {X 0,Y 213.721,Z 407.357,A -85,B 0,C 180,E1 -20741.124,E2 -20741.124} C_VEL
LIN {X 0,Y 213.709,Z 407.36,A -85,B 0,C 180,E1 -20743.678,E2 -20743.678} C_VEL
LIN {X 0,Y 213.704,Z 407.363,A -85,B 0,C 180,E1 -20746.345,E2 -20746.345} C_VEL
LIN {X 0,Y 213.761,Z 407.357,A -85,B 0,C 180,E1 -20750.209,E2 -20750.209} C_VEL
LIN {X 0,Y 214.793,Z 410.221,A -85,B 0,C 180,E1 -20750.583,E2 -20750.583} C_VEL
LIN {X 0,Y 216.615,Z 412.677,A -85,B 0,C 180,E1 -20751.084,E2 -20751.084} C_VEL
LIN {X 0,Y 219.86,Z 418.042,A -85,B 0,C 180,E1 -20751.987,E2 -20751.987} C_VEL
LIN {X 0,Y 225.726,Z 429.023,A -85,B 0,C 180,E1 -20753.577,E2 -20753.577} C_VEL
LIN {X 0,Y 232.786,Z 444.214,A -85,B 0,C 180,E1 -20755.418,E2 -20755.418} C_VEL
LIN {X 0,Y 236.869,Z 454.497,A -85,B 0,C 180,E1 -20756.469,E2 -20756.469} C_VEL
LIN {X 0,Y 234.82,Z 504.127,A -85,B 0,C 180,E1 -20757.911,E2 -20757.911} C_VEL
LIN {X 0,Y 234.031,Z 518.497,A -85,B 0,C 180,E1 -20758.441,E2 -20758.441} C_VEL
LIN {X 0,Y 232.605,Z 531.243,A -85,B 0,C 180,E1 -20759.219,E2 -20759.219} C_VEL
LIN {X 0,Y 230.767,Z 543.723,A -85,B 0,C 180,E1 -20760.338,E2 -20760.338} C_VEL
LIN {X 0,Y 228.562,Z 555.688,A -85,B 0,C 180,E1 -20761.786,E2 -20761.786} C_VEL
LIN {X 0,Y 226.121,Z 566.346,A -85,B 0,C 180,E1 -20763.463,E2 -20763.463} C_VEL
LIN {X 0,Y 223.651,Z 576.057,A -85,B 0,C 180,E1 -20765.395,E2 -20765.395} C_VEL
LIN {X 0,Y 221.291,Z 584.89,A -85,B 0,C 180,E1 -20767.598,E2 -20767.598} C_VEL
LIN {X 0,Y 218.658,Z 593.508,A -85,B 0,C 180,E1 -20770.276,E2 -20770.276} C_VEL
LIN {X 0,Y 216.381,Z 600.38,A -85,B 0,C 180,E1 -20773.004,E2 -20773.004} C_VEL
LIN {X 0,Y 214.66,Z 605.878,A -85,B 0,C 180,E1 -20775.786,E2 -20775.786} C_VEL
LIN {X 0,Y 213.296,Z 610.193,A -85,B 0,C 180,E1 -20778.598,E2 -20778.598} C_VEL
LIN {X 0,Y 212.646,Z 612.474,A -85,B 0,C 180,E1 -20780.488,E2 -20780.488} C_VEL
LIN {X 0,Y 212.162,Z 614.328,A -85,B 0,C 180,E1 -20782.386,E2 -20782.386} C_VEL
LIN {X 0,Y 211.774,Z 615.915,A -85,B 0,C 180,E1 -20784.619,E2 -20784.619} C_VEL
LIN {X 0,Y 211.544,Z 617.319,A -85,B 0,C 180,E1 -20788.096,E2 -20788.096} C_VEL
LIN {X 0,Y 211.521,Z 617.547,A -85,B 0,C 180,E1 -20790,E2 -20790} C_VEL
LIN {X 0,Y 211.544,Z 617.353,A -85,B 0,C 180,E1 -20791.904,E2 -20791.904} C_VEL
LIN {X 0,Y 211.775,Z 615.993,A -85,B 0,C 180,E1 -20795.381,E2 -20795.381} C_VEL
LIN {X 0,Y 212.165,Z 614.439,A -85,B 0,C 180,E1 -20797.615,E2 -20797.615} C_VEL
LIN {X 0,Y 212.972,Z 611.567,A -85,B 0,C 180,E1 -20800.457,E2 -20800.457} C_VEL
LIN {X 0,Y 214.128,Z 607.672,A -85,B 0,C 180,E1 -20803.283,E2 -20803.283} C_VEL
LIN {X 0,Y 215.704,Z 602.647,A -85,B 0,C 180,E1 -20806.078,E2 -20806.078} C_VEL
LIN {X 0,Y 217.785,Z 596.314,A -85,B 0,C 180,E1 -20808.827,E2 -20808.827} C_VEL
LIN {X 0,Y 220.331,Z 588.389,A -85,B 0,C 180,E1 -20811.52,E2 -20811.52} C_VEL
LIN {X 0,Y 222.694,Z 579.812,A -85,B 0,C 180,E1 -20813.867,E2 -20813.867} C_VEL
LIN {X 0,Y 225.125,Z 570.458,A -85,B 0,C 180,E1 -20815.917,E2 -20815.917} C_VEL
LIN {X 0,Y 227.829,Z 559.354,A -85,B 0,C 180,E1 -20817.813,E2 -20817.813} C_VEL
LIN {X 0,Y 230.06,Z 548.468,A -85,B 0,C 180,E1 -20819.261,E2 -20819.261} C_VEL
LIN {X 0,Y 232.046,Z 536.433,A -85,B 0,C 180,E1 -20820.485,E2 -20820.485} C_VEL
LIN {X 0,Y 233.576,Z 523.928,A -85,B 0,C 180,E1 -20821.402,E2 -20821.402} C_VEL
LIN {X 0,Y 234.64,Z 510.999,A -85,B 0,C 180,E1 -20821.997,E2 -20821.997} C_VEL
LIN {X 0,Y 236.978,Z 454.695,A -85,B 0,C 180,E1 -20823.651,E2 -20823.651} C_VEL
LIN {X 0,Y 231.188,Z 440.389,A -85,B 0,C 180,E1 -20825.149,E2 -20825.149} C_VEL
LIN {X 0,Y 223.983,Z 425.605,A -85,B 0,C 180,E1 -20827.045,E2 -20827.045} C_VEL
LIN {X 0,Y 218.338,Z 415.442,A -85,B 0,C 180,E1 -20828.596,E2 -20828.596} C_VEL
LIN {X 0,Y 215.778,Z 411.498,A -85,B 0,C 180,E1 -20829.31,E2 -20829.31} C_VEL
LIN {X 0,Y 214.139,Z 408.913,A -85,B 0,C 180,E1 -20829.782,E2 -20829.782} C_VEL
LIN {X 0,Y 213.765,Z 407.359,A -85,B 0,C 180,E1 -20829.954,E2 -20829.954} C_VEL
LIN {X 0,Y 213.711,Z 407.362,A -85,B 0,C 180,E1 -20833.678,E2 -20833.678} C_VEL
LIN {X 0,Y 213.751,Z 407.356,A -85,B 0,C 180,E1 -20836.332,E2 -20836.332} C_VEL
LIN {X 0,Y 213.74,Z 407.34,A -85,B 0,C 180,E1 -20841.337,E2 -20841.337} C_VEL
LIN {X 0,Y 213.773,Z 407.35,A -85,B 0,C 180,E1 -20846.021,E2 -20846.021} C_VEL
LIN {X 0,Y 213.785,Z 407.348,A -85,B 0,C 180,E1 -20850.454,E2 -20850.454} C_VEL
LIN {X 0,Y 213.808,Z 407.343,A -85,B 0,C 180,E1 -20854.702,E2 -20854.702} C_VEL
LIN {X 0,Y 213.845,Z 407.345,A -85,B 0,C 180,E1 -20858.807,E2 -20858.807} C_VEL
LIN {X 0,Y 213.949,Z 407.334,A -85,B 0,C 180,E1 -20862.804,E2 -20862.804} C_VEL
LIN {X 0,Y 213.985,Z 407.318,A -85,B 0,C 180,E1 -20866.708,E2 -20866.708} C_VEL
LIN {X 0,Y 214.201,Z 407.301,A -85,B 0,C 180,E1 -20870.558,E2 -20870.558} C_VEL
LIN {X 0,Y 214.117,Z 407.309,A -85,B 0,C 180,E1 -20874.349,E2 -20874.349} C_VEL
LIN {X 0,Y 214.451,Z 407.262,A -85,B 0,C 180,E1 -20878.122,E2 -20878.122} C_VEL
LIN {X 0,Y 214.555,Z 407.249,A -85,B 0,C 180,E1 -20880,E2 -20880} C_VEL
LIN {X 0,Y 214.45,Z 407.273,A -85,B 0,C 180,E1 -20881.878,E2 -20881.878} C_VEL
LIN {X 0,Y 214.199,Z 407.3,A -85,B 0,C 180,E1 -20887.541,E2 -20887.541} C_VEL
LIN {X 0,Y 214.003,Z 407.317,A -85,B 0,C 180,E1 -20891.364,E2 -20891.364} C_VEL
LIN {X 0,Y 213.939,Z 407.336,A -85,B 0,C 180,E1 -20895.236,E2 -20895.236} C_VEL
LIN {X 0,Y 213.844,Z 407.346,A -85,B 0,C 180,E1 -20899.187,E2 -20899.187} C_VEL
LIN {X 0,Y 213.851,Z 407.339,A -85,B 0,C 180,E1 -20903.227,E2 -20903.227} C_VEL
LIN {X 0,Y 213.832,Z 407.349,A -85,B 0,C 180,E1 -20907.449,E2 -20907.449} C_VEL
LIN {X 0,Y 213.77,Z 407.355,A -85,B 0,C 180,E1 -20911.737,E2 -20911.737} C_VEL
LIN {X 0,Y 213.746,Z 407.357,A -85,B 0,C 180,E1 -20916.288,E2 -20916.288} C_VEL
LIN {X 0,Y 213.715,Z 407.364,A -85,B 0,C 180,E1 -20921.125,E2 -20921.125} C_VEL
LIN {X 0,Y 213.711,Z 407.363,A -85,B 0,C 180,E1 -20924.213,E2 -20924.213} C_VEL
LIN {X 0,Y 213.373,Z 407.599,A -85,B 0,C 180,E1 -20924.965,E2 -20924.965} C_VEL
LIN {X 0,Y 212.534,Z 408.227,A -85,B 0,C 180,E1 -20925.679,E2 -20925.679} C_VEL
LIN {X 0,Y 210.291,Z 410.372,A -85,B 0,C 180,E1 -20927.015,E2 -20927.015} C_VEL
LIN {X 0,Y 208.714,Z 413.614,A -85,B 0,C 180,E1 -20928.286,E2 -20928.286} C_VEL
LIN {X 0,Y 208.986,Z 416.124,A -85,B 0,C 180,E1 -20929.008,E2 -20929.008} C_VEL
LIN {X 0,Y 209.499,Z 417.054,A -85,B 0,C 180,E1 -20929.222,E2 -20929.222} C_VEL
LIN {X 0,Y 211.888,Z 421.048,A -85,B 0,C 180,E1 -20929.948,E2 -20929.948} C_VEL
LIN {X 0,Y 218.048,Z 432.683,A -85,B 0,C 180,E1 -20931.767,E2 -20931.767} C_VEL
LIN {X 0,Y 224.251,Z 445.993,A -85,B 0,C 180,E1 -20933.519,E2 -20933.519} C_VEL
LIN {X 0,Y 228.735,Z 457.353,A -85,B 0,C 180,E1 -20934.769,E2 -20934.769} C_VEL
LIN {X 0,Y 230.506,Z 470.808,A -85,B 0,C 180,E1 -20935.576,E2 -20935.576} C_VEL
LIN {X 0,Y 228.083,Z 523.344,A -85,B 0,C 180,E1 -20937.164,E2 -20937.164} C_VEL
LIN {X 0,Y 226.657,Z 536.928,A -85,B 0,C 180,E1 -20937.89,E2 -20937.89} C_VEL
LIN {X 0,Y 224.745,Z 549.771,A -85,B 0,C 180,E1 -20938.937,E2 -20938.937} C_VEL
LIN {X 0,Y 222.507,Z 560.857,A -85,B 0,C 180,E1 -20940.166,E2 -20940.166} C_VEL
LIN {X 0,Y 219.82,Z 572.417,A -85,B 0,C 180,E1 -20941.862,E2 -20941.862} C_VEL
LIN {X 0,Y 217.013,Z 582.827,A -85,B 0,C 180,E1 -20943.816,E2 -20943.816} C_VEL
LIN {X 0,Y 214.504,Z 591.339,A -85,B 0,C 180,E1 -20945.823,E2 -20945.823} C_VEL
LIN {X 0,Y 212.333,Z 598.616,A -85,B 0,C 180,E1 -20947.937,E2 -20947.937} C_VEL
LIN {X 0,Y 210.12,Z 605.718,A -85,B 0,C 180,E1 -20950.459,E2 -20950.459} C_VEL
LIN {X 0,Y 208.056,Z 612.135,A -85,B 0,C 180,E1 -20953.314,E2 -20953.314} C_VEL
LIN {X 0,Y 206.367,Z 617.232,A -85,B 0,C 180,E1 -20956.208,E2 -20956.208} C_VEL
LIN {X 0,Y 205.324,Z 621.196,A -85,B 0,C 180,E1 -20959.148,E2 -20959.148} C_VEL
LIN {X 0,Y 204.642,Z 624.126,A -85,B 0,C 180,E1 -20962.104,E2 -20962.104} C_VEL
LIN {X 0,Y 204.397,Z 625.521,A -85,B 0,C 180,E1 -20964.079,E2 -20964.079} C_VEL
LIN {X 0,Y 204.297,Z 626.517,A -85,B 0,C 180,E1 -20966.054,E2 -20966.054} C_VEL
LIN {X 0,Y 204.325,Z 627.126,A -85,B 0,C 180,E1 -20968.028,E2 -20968.028} C_VEL
LIN {X 0,Y 204.392,Z 627.34,A -85,B 0,C 180,E1 -20970,E2 -20970} C_VEL
LIN {X 0,Y 204.325,Z 627.115,A -85,B 0,C 180,E1 -20971.971,E2 -20971.971} C_VEL
LIN {X 0,Y 204.402,Z 625.495,A -85,B 0,C 180,E1 -20975.92,E2 -20975.92} C_VEL
LIN {X 0,Y 204.642,Z 624.089,A -85,B 0,C 180,E1 -20977.895,E2 -20977.895} C_VEL
LIN {X 0,Y 205.323,Z 621.142,A -85,B 0,C 180,E1 -20980.851,E2 -20980.851} C_VEL
LIN {X 0,Y 206.362,Z 617.156,A -85,B 0,C 180,E1 -20983.792,E2 -20983.792} C_VEL
LIN {X 0,Y 208.348,Z 611.036,A -85,B 0,C 180,E1 -20987.167,E2 -20987.167} C_VEL
LIN {X 0,Y 210.529,Z 604.354,A -85,B 0,C 180,E1 -20990.009,E2 -20990.009} C_VEL
LIN {X 0,Y 213.086,Z 595.9,A -85,B 0,C 180,E1 -20992.857,E2 -20992.857} C_VEL
LIN {X 0,Y 215.588,Z 587.562,A -85,B 0,C 180,E1 -20995.074,E2 -20995.074} C_VEL
LIN {X 0,Y 218.501,Z 577.061,A -85,B 0,C 180,E1 -20997.28,E2 -20997.28} C_VEL
LIN {X 0,Y 221.469,Z 565.242,A -85,B 0,C 180,E1 -20999.203,E2 -20999.203} C_VEL
LIN {X 0,Y 223.979,Z 553.33,A -85,B 0,C 180,E1 -21000.656,E2 -21000.656} C_VEL
LIN {X 0,Y 225.826,Z 542.229,A -85,B 0,C 180,E1 -21001.68,E2 -21001.68} C_VEL
LIN {X 0,Y 227.589,Z 528.81,A -85,B 0,C 180,E1 -21002.533,E2 -21002.533} C_VEL
LIN {X 0,Y 228.484,Z 514.71,A -85,B 0,C 180,E1 -21003.086,E2 -21003.086} C_VEL
LIN {X 0,Y 230.286,Z 469.537,A -85,B 0,C 180,E1 -21004.45,E2 -21004.45} C_VEL
LIN {X 0,Y 228.529,Z 456.828,A -85,B 0,C 180,E1 -21005.227,E2 -21005.227} C_VEL
LIN {X 0,Y 222.719,Z 442.576,A -85,B 0,C 180,E1 -21006.841,E2 -21006.841} C_VEL
LIN {X 0,Y 215.719,Z 427.975,A -85,B 0,C 180,E1 -21008.844,E2 -21008.844} C_VEL
LIN {X 0,Y 210.511,Z 418.658,A -85,B 0,C 180,E1 -21010.394,E2 -21010.394} C_VEL
LIN {X 0,Y 208.317,Z 414.504,A -85,B 0,C 180,E1 -21011.124,E2 -21011.124} C_VEL
LIN {X 0,Y 206.616,Z 408.247,A -85,B 0,C 180,E1 -21014.998,E2 -21014.998} C_VEL
LIN {X 0,Y 206.661,Z 408.237,A -85,B 0,C 180,E1 -21019.749,E2 -21019.749} C_VEL
LIN {X 0,Y 206.699,Z 408.232,A -85,B 0,C 180,E1 -21024.689,E2 -21024.689} C_VEL
LIN {X 0,Y 206.707,Z 408.233,A -85,B 0,C 180,E1 -21029.336,E2 -21029.336} C_VEL
LIN {X 0,Y 206.736,Z 408.232,A -85,B 0,C 180,E1 -21033.772,E2 -21033.772} C_VEL
LIN {X 0,Y 206.779,Z 408.227,A -85,B 0,C 180,E1 -21038.046,E2 -21038.046} C_VEL
LIN {X 0,Y 206.88,Z 408.213,A -85,B 0,C 180,E1 -21042.197,E2 -21042.197} C_VEL
LIN {X 0,Y 206.897,Z 408.207,A -85,B 0,C 180,E1 -21046.245,E2 -21046.245} C_VEL
LIN {X 0,Y 207.1,Z 408.18,A -85,B 0,C 180,E1 -21050.231,E2 -21050.231} C_VEL
LIN {X 0,Y 207.061,Z 408.189,A -85,B 0,C 180,E1 -21054.156,E2 -21054.156} C_VEL
LIN {X 0,Y 207.383,Z 408.153,A -85,B 0,C 180,E1 -21058.058,E2 -21058.058} C_VEL
LIN {X 0,Y 207.517,Z 408.129,A -85,B 0,C 180,E1 -21060,E2 -21060} C_VEL
LIN {X 0,Y 207.386,Z 408.144,A -85,B 0,C 180,E1 -21061.942,E2 -21061.942} C_VEL
LIN {X 0,Y 207.191,Z 408.171,A -85,B 0,C 180,E1 -21067.798,E2 -21067.798} C_VEL
LIN {X 0,Y 206.985,Z 408.194,A -85,B 0,C 180,E1 -21071.755,E2 -21071.755} C_VEL
LIN {X 0,Y 206.869,Z 408.212,A -85,B 0,C 180,E1 -21075.771,E2 -21075.771} C_VEL
LIN {X 0,Y 206.815,Z 408.224,A -85,B 0,C 180,E1 -21079.866,E2 -21079.866} C_VEL
LIN {X 0,Y 206.77,Z 408.23,A -85,B 0,C 180,E1 -21084.072,E2 -21084.072} C_VEL
LIN {X 0,Y 206.745,Z 408.232,A -85,B 0,C 180,E1 -21088.419,E2 -21088.419} C_VEL
LIN {X 0,Y 206.711,Z 408.236,A -85,B 0,C 180,E1 -21092.956,E2 -21092.956} C_VEL
LIN {X 0,Y 206.723,Z 408.232,A -85,B 0,C 180,E1 -21095.32,E2 -21095.32} C_VEL
LIN {X 0,Y 206.67,Z 408.238,A -85,B 0,C 180,E1 -21100.249,E2 -21100.249} C_VEL
LIN {X 0,Y 206.635,Z 408.241,A -85,B 0,C 180,E1 -21104.419,E2 -21104.419} C_VEL
LIN {X 0,Y 206.66,Z 408.243,A -85,B 0,C 180,E1 -21108.577,E2 -21108.577} C_VEL
LIN {X 0,Y 207.687,Z 411.115,A -85,B 0,C 180,E1 -21108.982,E2 -21108.982} C_VEL
LIN {X 0,Y 209.747,Z 413.734,A -85,B 0,C 180,E1 -21109.588,E2 -21109.588} C_VEL
LIN {X 0,Y 215.236,Z 422.551,A -85,B 0,C 180,E1 -21111.201,E2 -21111.201} C_VEL
LIN {X 0,Y 221.648,Z 434.812,A -85,B 0,C 180,E1 -21113.02,E2 -21113.02} C_VEL
LIN {X 0,Y 228.64,Z 450.377,A -85,B 0,C 180,E1 -21114.926,E2 -21114.926} C_VEL
LIN {X 0,Y 230.926,Z 456.366,A -85,B 0,C 180,E1 -21115.548,E2 -21115.548} C_VEL
LIN {X 0,Y 228.832,Z 504.468,A -85,B 0,C 180,E1 -21116.971,E2 -21116.971} C_VEL
LIN {X 0,Y 227.975,Z 519.211,A -85,B 0,C 180,E1 -21117.535,E2 -21117.535} C_VEL
LIN {X 0,Y 226.387,Z 532.717,A -85,B 0,C 180,E1 -21118.408,E2 -21118.408} C_VEL
LIN {X 0,Y 224.631,Z 543.897,A -85,B 0,C 180,E1 -21119.442,E2 -21119.442} C_VEL
LIN {X 0,Y 222.329,Z 555.86,A -85,B 0,C 180,E1 -21120.921,E2 -21120.921} C_VEL
LIN {X 0,Y 219.778,Z 566.517,A -85,B 0,C 180,E1 -21122.634,E2 -21122.634} C_VEL
LIN {X 0,Y 217.205,Z 576.228,A -85,B 0,C 180,E1 -21124.614,E2 -21124.614} C_VEL
LIN {X 0,Y 214.725,Z 585.06,A -85,B 0,C 180,E1 -21126.874,E2 -21126.874} C_VEL
LIN {X 0,Y 211.973,Z 593.677,A -85,B 0,C 180,E1 -21129.627,E2 -21129.627} C_VEL
LIN {X 0,Y 209.59,Z 600.549,A -85,B 0,C 180,E1 -21132.435,E2 -21132.435} C_VEL
LIN {X 0,Y 207.78,Z 606.046,A -85,B 0,C 180,E1 -21135.305,E2 -21135.305} C_VEL
LIN {X 0,Y 206.346,Z 610.361,A -85,B 0,C 180,E1 -21138.209,E2 -21138.209} C_VEL
LIN {X 0,Y 205.655,Z 612.642,A -85,B 0,C 180,E1 -21140.162,E2 -21140.162} C_VEL
LIN {X 0,Y 205.12,Z 614.496,A -85,B 0,C 180,E1 -21142.123,E2 -21142.123} C_VEL
LIN {X 0,Y 204.674,Z 616.257,A -85,B 0,C 180,E1 -21144.742,E2 -21144.742} C_VEL
LIN {X 0,Y 204.45,Z 617.486,A -85,B 0,C 180,E1 -21148.03,E2 -21148.03} C_VEL
LIN {X 0,Y 204.424,Z 617.714,A -85,B 0,C 180,E1 -21150,E2 -21150} C_VEL
LIN {X 0,Y 204.449,Z 617.52,A -85,B 0,C 180,E1 -21151.97,E2 -21151.97} C_VEL
LIN {X 0,Y 204.674,Z 616.334,A -85,B 0,C 180,E1 -21155.258,E2 -21155.258} C_VEL
LIN {X 0,Y 205.123,Z 614.606,A -85,B 0,C 180,E1 -21157.878,E2 -21157.878} C_VEL
LIN {X 0,Y 205.973,Z 611.734,A -85,B 0,C 180,E1 -21160.817,E2 -21160.817} C_VEL
LIN {X 0,Y 207.228,Z 607.838,A -85,B 0,C 180,E1 -21163.734,E2 -21163.734} C_VEL
LIN {X 0,Y 208.885,Z 602.813,A -85,B 0,C 180,E1 -21166.618,E2 -21166.618} C_VEL
LIN {X 0,Y 211.071,Z 596.479,A -85,B 0,C 180,E1 -21169.45,E2 -21169.45} C_VEL
LIN {X 0,Y 213.723,Z 588.554,A -85,B 0,C 180,E1 -21172.22,E2 -21172.22} C_VEL
LIN {X 0,Y 216.12,Z 580.28,A -85,B 0,C 180,E1 -21174.553,E2 -21174.553} C_VEL
LIN {X 0,Y 218.768,Z 570.622,A -85,B 0,C 180,E1 -21176.729,E2 -21176.729} C_VEL
LIN {X 0,Y 221.579,Z 559.516,A -85,B 0,C 180,E1 -21178.668,E2 -21178.668} C_VEL
LIN {X 0,Y 223.903,Z 548.629,A -85,B 0,C 180,E1 -21180.147,E2 -21180.147} C_VEL
LIN {X 0,Y 225.974,Z 536.592,A -85,B 0,C 180,E1 -21181.396,E2 -21181.396} C_VEL
LIN {X 0,Y 227.592,Z 523.611,A -85,B 0,C 180,E1 -21182.36,E2 -21182.36} C_VEL
LIN {X 0,Y 228.723,Z 509.692,A -85,B 0,C 180,E1 -21182.991,E2 -21182.991} C_VEL
LIN {X 0,Y 231.042,Z 456.548,A -85,B 0,C 180,E1 -21184.574,E2 -21184.574} C_VEL
LIN {X 0,Y 225.565,Z 443.109,A -85,B 0,C 180,E1 -21186.061,E2 -21186.061} C_VEL
LIN {X 0,Y 218.09,Z 427.697,A -85,B 0,C 180,E1 -21188.143,E2 -21188.143} C_VEL
LIN {X 0,Y 213.742,Z 420.027,A -85,B 0,C 180,E1 -21189.395,E2 -21189.395} C_VEL
LIN {X 0,Y 209.547,Z 413.324,A -85,B 0,C 180,E1 -21190.645,E2 -21190.645} C_VEL
LIN {X 0,Y 207.274,Z 410.377,A -85,B 0,C 180,E1 -21191.323,E2 -21191.323} C_VEL
LIN {X 0,Y 206.649,Z 408.244,A -85,B 0,C 180,E1 -21191.62,E2 -21191.62} C_VEL
LIN {X 0,Y 206.663,Z 408.238,A -85,B 0,C 180,E1 -21195.574,E2 -21195.574} C_VEL
LIN {X 0,Y 206.675,Z 408.217,A -85,B 0,C 180,E1 -21199.752,E2 -21199.752} C_VEL
LIN {X 0,Y 206.735,Z 408.231,A -85,B 0,C 180,E1 -21204.695,E2 -21204.695} C_VEL
LIN {X 0,Y 206.727,Z 408.231,A -85,B 0,C 180,E1 -21209.339,E2 -21209.339} C_VEL
LIN {X 0,Y 206.738,Z 408.23,A -85,B 0,C 180,E1 -21213.773,E2 -21213.773} C_VEL
LIN {X 0,Y 206.783,Z 408.229,A -85,B 0,C 180,E1 -21218.046,E2 -21218.046} C_VEL
LIN {X 0,Y 206.882,Z 408.21,A -85,B 0,C 180,E1 -21222.197,E2 -21222.197} C_VEL
LIN {X 0,Y 206.918,Z 408.198,A -85,B 0,C 180,E1 -21226.246,E2 -21226.246} C_VEL
LIN {X 0,Y 207.137,Z 408.182,A -85,B 0,C 180,E1 -21230.233,E2 -21230.233} C_VEL
LIN {X 0,Y 207.08,Z 408.182,A -85,B 0,C 180,E1 -21234.156,E2 -21234.156} C_VEL
LIN {X 0,Y 207.387,Z 408.142,A -85,B 0,C 180,E1 -21238.058,E2 -21238.058} C_VEL
LIN {X 0,Y 207.519,Z 408.124,A -85,B 0,C 180,E1 -21240,E2 -21240} C_VEL
LIN {X 0,Y 207.386,Z 408.153,A -85,B 0,C 180,E1 -21241.942,E2 -21241.942} C_VEL
LIN {X 0,Y 207.141,Z 408.181,A -85,B 0,C 180,E1 -21247.8,E2 -21247.8} C_VEL
LIN {X 0,Y 206.929,Z 408.197,A -85,B 0,C 180,E1 -21251.758,E2 -21251.758} C_VEL
LIN {X 0,Y 206.872,Z 408.211,A -85,B 0,C 180,E1 -21255.77,E2 -21255.77} C_VEL
LIN {X 0,Y 206.788,Z 408.227,A -85,B 0,C 180,E1 -21259.869,E2 -21259.869} C_VEL
LIN {X 0,Y 206.767,Z 408.229,A -85,B 0,C 180,E1 -21264.072,E2 -21264.072} C_VEL
LIN {X 0,Y 206.74,Z 408.23,A -85,B 0,C 180,E1 -21268.419,E2 -21268.419} C_VEL
LIN {X 0,Y 206.701,Z 408.235,A -85,B 0,C 180,E1 -21272.957,E2 -21272.957} C_VEL
LIN {X 0,Y 206.682,Z 408.238,A -85,B 0,C 180,E1 -21277.739,E2 -21277.739} C_VEL
LIN {X 0,Y 206.645,Z 408.243,A -85,B 0,C 180,E1 -21281.563,E2 -21281.563} C_VEL
LIN {X 0,Y 206.726,Z 408.355,A -85,B 0,C 180,E1 -21285.065,E2 -21285.065} C_VEL
LIN {X 0,Y 208.402,Z 414.695,A -85,B 0,C 180,E1 -21288.858,E2 -21288.858} C_VEL
LIN {X 0,Y 209.499,Z 417.054,A -85,B 0,C 180,E1 -21289.222,E2 -21289.222} C_VEL
LIN {X 0,Y 211.174,Z 420.031,A -85,B 0,C 180,E1 -21289.741,E2 -21289.741} C_VEL
LIN {X 0,Y 212.412,Z 423.405,A -85,B 0,C 180,E1 -21290.167,E2 -21290.167} C_VEL
LIN {X 0,Y 214.021,Z 430.767,A -85,B 0,C 180,E1 -21290.836,E2 -21290.836} C_VEL
LIN {X 0,Y 216.193,Z 442.171,A -85,B 0,C 180,E1 -21291.774,E2 -21291.774} C_VEL
LIN {X 0,Y 217.404,Z 445.707,A -85,B 0,C 180,E1 -21292.168,E2 -21292.168} C_VEL
LIN {X 0,Y 223.009,Z 459.444,A -85,B 0,C 180,E1 -21293.811,E2 -21293.811} C_VEL
LIN {X 0,Y 224.607,Z 471.826,A -85,B 0,C 180,E1 -21294.583,E2 -21294.583} C_VEL
LIN {X 0,Y 222.177,Z 523.081,A -85,B 0,C 180,E1 -21296.169,E2 -21296.169} C_VEL
LIN {X 0,Y 220.671,Z 536.911,A -85,B 0,C 180,E1 -21296.922,E2 -21296.922} C_VEL
LIN {X 0,Y 218.886,Z 548.503,A -85,B 0,C 180,E1 -21297.873,E2 -21297.873} C_VEL
LIN {X 0,Y 216.362,Z 560.694,A -85,B 0,C 180,E1 -21299.229,E2 -21299.229} C_VEL
LIN {X 0,Y 213.582,Z 572.253,A -85,B 0,C 180,E1 -21300.964,E2 -21300.964} C_VEL
LIN {X 0,Y 210.676,Z 582.663,A -85,B 0,C 180,E1 -21302.965,E2 -21302.965} C_VEL
LIN {X 0,Y 208.032,Z 591.174,A -85,B 0,C 180,E1 -21305.02,E2 -21305.02} C_VEL
LIN {X 0,Y 205.519,Z 599.141,A -85,B 0,C 180,E1 -21307.414,E2 -21307.414} C_VEL
LIN {X 0,Y 203.428,Z 605.552,A -85,B 0,C 180,E1 -21309.788,E2 -21309.788} C_VEL
LIN {X 0,Y 201.22,Z 611.968,A -85,B 0,C 180,E1 -21312.729,E2 -21312.729} C_VEL
LIN {X 0,Y 199.438,Z 617.065,A -85,B 0,C 180,E1 -21315.719,E2 -21315.719} C_VEL
LIN {X 0,Y 198.313,Z 621.029,A -85,B 0,C 180,E1 -21318.76,E2 -21318.76} C_VEL
LIN {X 0,Y 197.593,Z 623.959,A -85,B 0,C 180,E1 -21321.82,E2 -21321.82} C_VEL
LIN {X 0,Y 197.338,Z 625.354,A -85,B 0,C 180,E1 -21323.866,E2 -21323.866} C_VEL
LIN {X 0,Y 197.232,Z 626.959,A -85,B 0,C 180,E1 -21327.958,E2 -21327.958} C_VEL
LIN {X 0,Y 197.296,Z 627.173,A -85,B 0,C 180,E1 -21330,E2 -21330} C_VEL
LIN {X 0,Y 197.201,Z 626.475,A -85,B 0,C 180,E1 -21333.724,E2 -21333.724} C_VEL
LIN {X 0,Y 197.341,Z 625.328,A -85,B 0,C 180,E1 -21336.133,E2 -21336.133} C_VEL
LIN {X 0,Y 197.592,Z 623.921,A -85,B 0,C 180,E1 -21338.179,E2 -21338.179} C_VEL
LIN {X 0,Y 198.312,Z 620.973,A -85,B 0,C 180,E1 -21341.239,E2 -21341.239} C_VEL
LIN {X 0,Y 199.433,Z 616.987,A -85,B 0,C 180,E1 -21344.281,E2 -21344.281} C_VEL
LIN {X 0,Y 201.563,Z 610.867,A -85,B 0,C 180,E1 -21347.763,E2 -21347.763} C_VEL
LIN {X 0,Y 203.866,Z 604.185,A -85,B 0,C 180,E1 -21350.692,E2 -21350.692} C_VEL
LIN {X 0,Y 206.423,Z 596.042,A -85,B 0,C 180,E1 -21353.528,E2 -21353.528} C_VEL
LIN {X 0,Y 209.152,Z 587.392,A -85,B 0,C 180,E1 -21355.902,E2 -21355.902} C_VEL
LIN {X 0,Y 212.227,Z 576.891,A -85,B 0,C 180,E1 -21358.157,E2 -21358.157} C_VEL
LIN {X 0,Y 215.286,Z 565.07,A -85,B 0,C 180,E1 -21360.127,E2 -21360.127} C_VEL
LIN {X 0,Y 217.9,Z 553.157,A -85,B 0,C 180,E1 -21361.609,E2 -21361.609} C_VEL
LIN {X 0,Y 219.835,Z 542.055,A -85,B 0,C 180,E1 -21362.648,E2 -21362.648} C_VEL
LIN {X 0,Y 221.586,Z 529.135,A -85,B 0,C 180,E1 -21363.491,E2 -21363.491} C_VEL
LIN {X 0,Y 222.501,Z 516.296,A -85,B 0,C 180,E1 -21364.028,E2 -21364.028} C_VEL
LIN {X 0,Y 224.426,Z 470.493,A -85,B 0,C 180,E1 -21365.439,E2 -21365.439} C_VEL
LIN {X 0,Y 222.901,Z 459.411,A -85,B 0,C 180,E1 -21366.147,E2 -21366.147} C_VEL
LIN {X 0,Y 217.38,Z 445.663,A -85,B 0,C 180,E1 -21367.769,E2 -21367.769} C_VEL
LIN {X 0,Y 210.516,Z 431.376,A -85,B 0,C 180,E1 -21369.839,E2 -21369.839} C_VEL
LIN {X 0,Y 205.837,Z 422.921,A -85,B 0,C 180,E1 -21371.309,E2 -21371.309} C_VEL
LIN {X 0,Y 203.078,Z 418.192,A -85,B 0,C 180,E1 -21372.213,E2 -21372.213} C_VEL
LIN {X 0,Y 201.029,Z 414.342,A -85,B 0,C 180,E1 -21372.929,E2 -21372.929} C_VEL
LIN {X 0,Y 199.567,Z 409.12,A -85,B 0,C 180,E1 -21376.388,E2 -21376.388} C_VEL
LIN {X 0,Y 199.612,Z 409.119,A -85,B 0,C 180,E1 -21380.767,E2 -21380.767} C_VEL
LIN {X 0,Y 199.612,Z 409.114,A -85,B 0,C 180,E1 -21385.713,E2 -21385.713} C_VEL
LIN {X 0,Y 199.694,Z 409.106,A -85,B 0,C 180,E1 -21388.136,E2 -21388.136} C_VEL
LIN {X 0,Y 199.687,Z 409.106,A -85,B 0,C 180,E1 -21392.772,E2 -21392.772} C_VEL
LIN {X 0,Y 199.751,Z 409.1,A -85,B 0,C 180,E1 -21397.231,E2 -21397.231} C_VEL
LIN {X 0,Y 199.839,Z 409.089,A -85,B 0,C 180,E1 -21401.722,E2 -21401.722} C_VEL
LIN {X 0,Y 199.838,Z 409.083,A -85,B 0,C 180,E1 -21405.748,E2 -21405.748} C_VEL
LIN {X 0,Y 200.023,Z 409.061,A -85,B 0,C 180,E1 -21409.882,E2 -21409.882} C_VEL
LIN {X 0,Y 200.022,Z 409.067,A -85,B 0,C 180,E1 -21413.949,E2 -21413.949} C_VEL
LIN {X 0,Y 200.323,Z 409.032,A -85,B 0,C 180,E1 -21417.99,E2 -21417.99} C_VEL
LIN {X 0,Y 200.481,Z 409.005,A -85,B 0,C 180,E1 -21420,E2 -21420} C_VEL
LIN {X 0,Y 200.037,Z 409.069,A -85,B 0,C 180,E1 -21424.029,E2 -21424.029} C_VEL
LIN {X 0,Y 200.134,Z 409.052,A -85,B 0,C 180,E1 -21428.075,E2 -21428.075} C_VEL
LIN {X 0,Y 199.916,Z 409.074,A -85,B 0,C 180,E1 -21432.177,E2 -21432.177} C_VEL
LIN {X 0,Y 199.808,Z 409.087,A -85,B 0,C 180,E1 -21436.343,E2 -21436.343} C_VEL
LIN {X 0,Y 199.743,Z 409.101,A -85,B 0,C 180,E1 -21440.601,E2 -21440.601} C_VEL
LIN {X 0,Y 199.677,Z 409.111,A -85,B 0,C 180,E1 -21444.984,E2 -21444.984} C_VEL
LIN {X 0,Y 199.676,Z 409.109,A -85,B 0,C 180,E1 -21449.522,E2 -21449.522} C_VEL
LIN {X 0,Y 199.666,Z 409.113,A -85,B 0,C 180,E1 -21452.353,E2 -21452.353} C_VEL
LIN {X 0,Y 199.641,Z 409.114,A -85,B 0,C 180,E1 -21456.76,E2 -21456.76} C_VEL
LIN {X 0,Y 199.64,Z 409.116,A -85,B 0,C 180,E1 -21459.321,E2 -21459.321} C_VEL
LIN {X 0,Y 199.58,Z 409.124,A -85,B 0,C 180,E1 -21462.312,E2 -21462.312} C_VEL
LIN {X 0,Y 199.578,Z 409.12,A -85,B 0,C 180,E1 -21466.773,E2 -21466.773} C_VEL
LIN {X 0,Y 200.692,Z 412.149,A -85,B 0,C 180,E1 -21467.258,E2 -21467.258} C_VEL
LIN {X 0,Y 202.736,Z 414.638,A -85,B 0,C 180,E1 -21467.91,E2 -21467.91} C_VEL
LIN {X 0,Y 204.949,Z 417.919,A -85,B 0,C 180,E1 -21468.621,E2 -21468.621} C_VEL
LIN {X 0,Y 210.764,Z 427.237,A -85,B 0,C 180,E1 -21470.414,E2 -21470.414} C_VEL
LIN {X 0,Y 216.901,Z 439.207,A -85,B 0,C 180,E1 -21472.244,E2 -21472.244} C_VEL
LIN {X 0,Y 223.737,Z 454.806,A -85,B 0,C 180,E1 -21474.206,E2 -21474.206} C_VEL
LIN {X 0,Y 224.997,Z 458.122,A -85,B 0,C 180,E1 -21474.566,E2 -21474.566} C_VEL
LIN {X 0,Y 222.965,Z 503.923,A -85,B 0,C 180,E1 -21475.958,E2 -21475.958} C_VEL
LIN {X 0,Y 222.05,Z 519.124,A -85,B 0,C 180,E1 -21476.539,E2 -21476.539} C_VEL
LIN {X 0,Y 220.568,Z 531.594,A -85,B 0,C 180,E1 -21477.338,E2 -21477.338} C_VEL
LIN {X 0,Y 218.556,Z 544.07,A -85,B 0,C 180,E1 -21478.497,E2 -21478.497} C_VEL
LIN {X 0,Y 216.158,Z 556.032,A -85,B 0,C 180,E1 -21480.007,E2 -21480.007} C_VEL
LIN {X 0,Y 213.506,Z 566.688,A -85,B 0,C 180,E1 -21481.759,E2 -21481.759} C_VEL
LIN {X 0,Y 210.807,Z 576.399,A -85,B 0,C 180,E1 -21483.786,E2 -21483.786} C_VEL
LIN {X 0,Y 208.201,Z 585.231,A -85,B 0,C 180,E1 -21486.105,E2 -21486.105} C_VEL
LIN {X 0,Y 205.811,Z 592.518,A -85,B 0,C 180,E1 -21488.464,E2 -21488.464} C_VEL
LIN {X 0,Y 203.243,Z 599.69,A -85,B 0,C 180,E1 -21491.346,E2 -21491.346} C_VEL
LIN {X 0,Y 201.533,Z 604.523,A -85,B 0,C 180,E1 -21493.801,E2 -21493.801} C_VEL
LIN {X 0,Y 199.85,Z 609.219,A -85,B 0,C 180,E1 -21496.787,E2 -21496.787} C_VEL
LIN {X 0,Y 198.656,Z 612.81,A -85,B 0,C 180,E1 -21499.812,E2 -21499.812} C_VEL
LIN {X 0,Y 198.078,Z 614.664,A -85,B 0,C 180,E1 -21501.841,E2 -21501.841} C_VEL
LIN {X 0,Y 197.568,Z 616.613,A -85,B 0,C 180,E1 -21504.899,E2 -21504.899} C_VEL
LIN {X 0,Y 197.358,Z 617.653,A -85,B 0,C 180,E1 -21507.96,E2 -21507.96} C_VEL
LIN {X 0,Y 197.329,Z 617.881,A -85,B 0,C 180,E1 -21510,E2 -21510} C_VEL
LIN {X 0,Y 197.358,Z 617.687,A -85,B 0,C 180,E1 -21512.041,E2 -21512.041} C_VEL
LIN {X 0,Y 197.583,Z 616.661,A -85,B 0,C 180,E1 -21515.152,E2 -21515.152} C_VEL
LIN {X 0,Y 198.082,Z 614.773,A -85,B 0,C 180,E1 -21518.159,E2 -21518.159} C_VEL
LIN {X 0,Y 199.001,Z 611.9,A -85,B 0,C 180,E1 -21521.201,E2 -21521.201} C_VEL
LIN {X 0,Y 200.33,Z 608.004,A -85,B 0,C 180,E1 -21524.216,E2 -21524.216} C_VEL
LIN {X 0,Y 202.067,Z 602.979,A -85,B 0,C 180,E1 -21527.196,E2 -21527.196} C_VEL
LIN {X 0,Y 204.388,Z 596.644,A -85,B 0,C 180,E1 -21530.113,E2 -21530.113} C_VEL
LIN {X 0,Y 207.15,Z 588.719,A -85,B 0,C 180,E1 -21532.965,E2 -21532.965} C_VEL
LIN {X 0,Y 209.59,Z 580.733,A -85,B 0,C 180,E1 -21535.285,E2 -21535.285} C_VEL
LIN {X 0,Y 212.434,Z 570.786,A -85,B 0,C 180,E1 -21537.592,E2 -21537.592} C_VEL
LIN {X 0,Y 215.382,Z 559.678,A -85,B 0,C 180,E1 -21539.574,E2 -21539.574} C_VEL
LIN {X 0,Y 217.79,Z 548.79,A -85,B 0,C 180,E1 -21541.086,E2 -21541.086} C_VEL
LIN {X 0,Y 219.951,Z 536.752,A -85,B 0,C 180,E1 -21542.359,E2 -21542.359} C_VEL
LIN {X 0,Y 221.607,Z 524.122,A -85,B 0,C 180,E1 -21543.319,E2 -21543.319} C_VEL
LIN {X 0,Y 222.753,Z 511.108,A -85,B 0,C 180,E1 -21543.936,E2 -21543.936} C_VEL
LIN {X 0,Y 225.141,Z 458.332,A -85,B 0,C 180,E1 -21545.552,E2 -21545.552} C_VEL
LIN {X 0,Y 220.034,Z 445.883,A -85,B 0,C 180,E1 -21547.011,E2 -21547.011} C_VEL
LIN {X 0,Y 213.193,Z 431.686,A -85,B 0,C 180,E1 -21549.019,E2 -21549.019} C_VEL
LIN {X 0,Y 208.838,Z 423.949,A -85,B 0,C 180,E1 -21550.341,E2 -21550.341} C_VEL
LIN {X 0,Y 204.518,Z 417.409,A -85,B 0,C 180,E1 -21551.683,E2 -21551.683} C_VEL
LIN {X 0,Y 202.129,Z 413.745,A -85,B 0,C 180,E1 -21552.465,E2 -21552.465} C_VEL
LIN {X 0,Y 200.217,Z 411.267,A -85,B 0,C 180,E1 -21553.09,E2 -21553.09} C_VEL
LIN {X 0,Y 199.583,Z 409.121,A -85,B 0,C 180,E1 -21553.389,E2 -21553.389} C_VEL
LIN {X 0,Y 199.603,Z 409.117,A -85,B 0,C 180,E1 -21558.011,E2 -21558.011} C_VEL
LIN {X 0,Y 199.645,Z 409.09,A -85,B 0,C 180,E1 -21560.757,E2 -21560.757} C_VEL
LIN {X 0,Y 199.638,Z 409.111,A -85,B 0,C 180,E1 -21565.718,E2 -21565.718} C_VEL
LIN {X 0,Y 199.708,Z 409.11,A -85,B 0,C 180,E1 -21568.138,E2 -21568.138} C_VEL
LIN {X 0,Y 199.692,Z 409.111,A -85,B 0,C 180,E1 -21572.772,E2 -21572.772} C_VEL
LIN {X 0,Y 199.754,Z 409.102,A -85,B 0,C 180,E1 -21577.231,E2 -21577.231} C_VEL
LIN {X 0,Y 199.842,Z 409.084,A -85,B 0,C 180,E1 -21581.722,E2 -21581.722} C_VEL
LIN {X 0,Y 199.853,Z 409.08,A -85,B 0,C 180,E1 -21585.749,E2 -21585.749} C_VEL
LIN {X 0,Y 200.08,Z 409.063,A -85,B 0,C 180,E1 -21589.885,E2 -21589.885} C_VEL
LIN {X 0,Y 200.043,Z 409.057,A -85,B 0,C 180,E1 -21593.95,E2 -21593.95} C_VEL
LIN {X 0,Y 200.327,Z 409.021,A -85,B 0,C 180,E1 -21597.989,E2 -21597.989} C_VEL
LIN {X 0,Y 200.484,Z 409,A -85,B 0,C 180,E1 -21600,E2 -21600} C_VEL
LIN {X 0,Y 200.032,Z 409.061,A -85,B 0,C 180,E1 -21604.029,E2 -21604.029} C_VEL
LIN {X 0,Y 200.09,Z 409.062,A -85,B 0,C 180,E1 -21608.077,E2 -21608.077} C_VEL
LIN {X 0,Y 199.879,Z 409.076,A -85,B 0,C 180,E1 -21612.179,E2 -21612.179} C_VEL
LIN {X 0,Y 199.809,Z 409.088,A -85,B 0,C 180,E1 -21616.343,E2 -21616.343} C_VEL
LIN {X 0,Y 199.704,Z 409.108,A -85,B 0,C 180,E1 -21620.605,E2 -21620.605} C_VEL
LIN {X 0,Y 199.676,Z 409.113,A -85,B 0,C 180,E1 -21624.984,E2 -21624.984} C_VEL
LIN {X 0,Y 199.667,Z 409.113,A -85,B 0,C 180,E1 -21629.523,E2 -21629.523} C_VEL
LIN {X 0,Y 199.674,Z 409.11,A -85,B 0,C 180,E1 -21632.355,E2 -21632.355} C_VEL
LIN {X 0,Y 199.626,Z 409.116,A -85,B 0,C 180,E1 -21636.763,E2 -21636.763} C_VEL
LIN {X 0,Y 199.611,Z 409.12,A -85,B 0,C 180,E1 -21639.328,E2 -21639.328} C_VEL
LIN {X 0,Y 199.602,Z 409.158,A -85,B 0,C 180,E1 -21643.603,E2 -21643.603} C_VEL
LIN {X 0,Y 201.038,Z 414.383,A -85,B 0,C 180,E1 -21646.992,E2 -21646.992} C_VEL
LIN {X 0,Y 203.443,Z 418.695,A -85,B 0,C 180,E1 -21647.819,E2 -21647.819} C_VEL
LIN {X 0,Y 209.773,Z 429.983,A -85,B 0,C 180,E1 -21649.855,E2 -21649.855} C_VEL
LIN {X 0,Y 216.718,Z 444.131,A -85,B 0,C 180,E1 -21651.963,E2 -21651.963} C_VEL
LIN {X 0,Y 217.404,Z 445.707,A -85,B 0,C 180,E1 -21652.168,E2 -21652.168} C_VEL
LIN {X 0,Y 218.334,Z 449.307,A -85,B 0,C 180,E1 -21652.503,E2 -21652.503} C_VEL
LIN {X 0,Y 218.454,Z 455.847,A -85,B 0,C 180,E1 -21652.791,E2 -21652.791} C_VEL
LIN {X 0,Y 218.076,Z 465.32,A -85,B 0,C 180,E1 -21653.099,E2 -21653.099} C_VEL
LIN {X 0,Y 218.186,Z 466.646,A -85,B 0,C 180,E1 -21653.174,E2 -21653.174} C_VEL
LIN {X 0,Y 218.787,Z 473.228,A -85,B 0,C 180,E1 -21653.554,E2 -21653.554} C_VEL
LIN {X 0,Y 216.319,Z 522.888,A -85,B 0,C 180,E1 -21655.12,E2 -21655.12} C_VEL
LIN {X 0,Y 214.848,Z 536.255,A -85,B 0,C 180,E1 -21655.859,E2 -21655.859} C_VEL
LIN {X 0,Y 212.906,Z 548.342,A -85,B 0,C 180,E1 -21656.857,E2 -21656.857} C_VEL
LIN {X 0,Y 210.286,Z 560.532,A -85,B 0,C 180,E1 -21658.238,E2 -21658.238} C_VEL
LIN {X 0,Y 207.383,Z 572.09,A -85,B 0,C 180,E1 -21660.008,E2 -21660.008} C_VEL
LIN {X 0,Y 204.371,Z 582.499,A -85,B 0,C 180,E1 -21662.06,E2 -21662.06} C_VEL
LIN {X 0,Y 201.601,Z 591.01,A -85,B 0,C 180,E1 -21664.166,E2 -21664.166} C_VEL
LIN {X 0,Y 198.706,Z 599.654,A -85,B 0,C 180,E1 -21666.866,E2 -21666.866} C_VEL
LIN {X 0,Y 196.318,Z 606.54,A -85,B 0,C 180,E1 -21669.571,E2 -21669.571} C_VEL
LIN {X 0,Y 194.427,Z 611.802,A -85,B 0,C 180,E1 -21672.106,E2 -21672.106} C_VEL
LIN {X 0,Y 192.531,Z 616.898,A -85,B 0,C 180,E1 -21675.195,E2 -21675.195} C_VEL
LIN {X 0,Y 191.322,Z 620.862,A -85,B 0,C 180,E1 -21678.343,E2 -21678.343} C_VEL
LIN {X 0,Y 190.543,Z 623.792,A -85,B 0,C 180,E1 -21681.515,E2 -21681.515} C_VEL
LIN {X 0,Y 190.277,Z 625.187,A -85,B 0,C 180,E1 -21683.638,E2 -21683.638} C_VEL
LIN {X 0,Y 190.141,Z 626.793,A -85,B 0,C 180,E1 -21687.881,E2 -21687.881} C_VEL
LIN {X 0,Y 190.202,Z 627.006,A -85,B 0,C 180,E1 -21690,E2 -21690} C_VEL
LIN {X 0,Y 190.116,Z 626.436,A -85,B 0,C 180,E1 -21693.525,E2 -21693.525} C_VEL
LIN {X 0,Y 190.279,Z 625.16,A -85,B 0,C 180,E1 -21696.361,E2 -21696.361} C_VEL
LIN {X 0,Y 190.542,Z 623.752,A -85,B 0,C 180,E1 -21698.484,E2 -21698.484} C_VEL
LIN {X 0,Y 191.321,Z 620.804,A -85,B 0,C 180,E1 -21701.656,E2 -21701.656} C_VEL
LIN {X 0,Y 192.526,Z 616.818,A -85,B 0,C 180,E1 -21704.805,E2 -21704.805} C_VEL
LIN {X 0,Y 194.803,Z 610.698,A -85,B 0,C 180,E1 -21708.401,E2 -21708.401} C_VEL
LIN {X 0,Y 197.225,Z 604.04,A -85,B 0,C 180,E1 -21711.412,E2 -21711.412} C_VEL
LIN {X 0,Y 199.911,Z 595.872,A -85,B 0,C 180,E1 -21714.343,E2 -21714.343} C_VEL
LIN {X 0,Y 202.764,Z 587.221,A -85,B 0,C 180,E1 -21716.782,E2 -21716.782} C_VEL
LIN {X 0,Y 206.003,Z 576.721,A -85,B 0,C 180,E1 -21719.088,E2 -21719.088} C_VEL
LIN {X 0,Y 209.184,Z 564.899,A -85,B 0,C 180,E1 -21721.101,E2 -21721.101} C_VEL
LIN {X 0,Y 211.881,Z 552.984,A -85,B 0,C 180,E1 -21722.616,E2 -21722.616} C_VEL
LIN {X 0,Y 213.901,Z 541.88,A -85,B 0,C 180,E1 -21723.673,E2 -21723.673} C_VEL
LIN {X 0,Y 215.673,Z 528.72,A -85,B 0,C 180,E1 -21724.555,E2 -21724.555} C_VEL
LIN {X 0,Y 216.7,Z 514.989,A -85,B 0,C 180,E1 -21725.114,E2 -21725.114} C_VEL
LIN {X 0,Y 218.595,Z 470.938,A -85,B 0,C 180,E1 -21726.508,E2 -21726.508} C_VEL
LIN {X 0,Y 217.326,Z 461.843,A -85,B 0,C 180,E1 -21727.122,E2 -21727.122} C_VEL
LIN {X 0,Y 211.183,Z 446.811,A -85,B 0,C 180,E1 -21729.026,E2 -21729.026} C_VEL
LIN {X 0,Y 204.406,Z 432.797,A -85,B 0,C 180,E1 -21731.208,E2 -21731.208} C_VEL
LIN {X 0,Y 198.389,Z 422.319,A -85,B 0,C 180,E1 -21733.245,E2 -21733.245} C_VEL
LIN {X 0,Y 196.306,Z 418.657,A -85,B 0,C 180,E1 -21733.997,E2 -21733.997} C_VEL
LIN {X 0,Y 193.822,Z 414.622,A -85,B 0,C 180,E1 -21734.911,E2 -21734.911} C_VEL
LIN {X 0,Y 193.588,Z 413.937,A -85,B 0,C 180,E1 -21735.117,E2 -21735.117} C_VEL
LIN {X 0,Y 192.537,Z 410.001,A -85,B 0,C 180,E1 -21737.947,E2 -21737.947} C_VEL
LIN {X 0,Y 192.587,Z 409.993,A -85,B 0,C 180,E1 -21743.402,E2 -21743.402} C_VEL
LIN {X 0,Y 192.608,Z 409.992,A -85,B 0,C 180,E1 -21747.059,E2 -21747.059} C_VEL
LIN {X 0,Y 192.661,Z 409.982,A -85,B 0,C 180,E1 -21751.691,E2 -21751.691} C_VEL
LIN {X 0,Y 192.713,Z 409.973,A -85,B 0,C 180,E1 -21756.35,E2 -21756.35} C_VEL
LIN {X 0,Y 192.783,Z 409.966,A -85,B 0,C 180,E1 -21761.413,E2 -21761.413} C_VEL
LIN {X 0,Y 192.766,Z 409.963,A -85,B 0,C 180,E1 -21765.214,E2 -21765.214} C_VEL
LIN {X 0,Y 192.946,Z 409.944,A -85,B 0,C 180,E1 -21769.567,E2 -21769.567} C_VEL
LIN {X 0,Y 192.984,Z 409.946,A -85,B 0,C 180,E1 -21773.728,E2 -21773.728} C_VEL
LIN {X 0,Y 193.264,Z 409.911,A -85,B 0,C 180,E1 -21777.916,E2 -21777.916} C_VEL
LIN {X 0,Y 193.445,Z 409.881,A -85,B 0,C 180,E1 -21780,E2 -21780} C_VEL
LIN {X 0,Y 192.984,Z 409.946,A -85,B 0,C 180,E1 -21784.177,E2 -21784.177} C_VEL
LIN {X 0,Y 193.081,Z 409.933,A -85,B 0,C 180,E1 -21788.372,E2 -21788.372} C_VEL
LIN {X 0,Y 192.855,Z 409.955,A -85,B 0,C 180,E1 -21792.63,E2 -21792.63} C_VEL
LIN {X 0,Y 192.783,Z 409.97,A -85,B 0,C 180,E1 -21798.587,E2 -21798.587} C_VEL
LIN {X 0,Y 192.67,Z 409.985,A -85,B 0,C 180,E1 -21804.228,E2 -21804.228} C_VEL
LIN {X 0,Y 192.651,Z 409.987,A -85,B 0,C 180,E1 -21808.892,E2 -21808.892} C_VEL
LIN {X 0,Y 192.601,Z 409.99,A -85,B 0,C 180,E1 -21813.186,E2 -21813.186} C_VEL
LIN {X 0,Y 192.611,Z 409.991,A -85,B 0,C 180,E1 -21816.608,E2 -21816.608} C_VEL
LIN {X 0,Y 192.526,Z 409.996,A -85,B 0,C 180,E1 -21821.077,E2 -21821.077} C_VEL
LIN {X 0,Y 192.536,Z 409.998,A -85,B 0,C 180,E1 -21824.84,E2 -21824.84} C_VEL
LIN {X 0,Y 193.538,Z 412.852,A -85,B 0,C 180,E1 -21825.291,E2 -21825.291} C_VEL
LIN {X 0,Y 195.759,Z 415.534,A -85,B 0,C 180,E1 -21826.07,E2 -21826.07} C_VEL
LIN {X 0,Y 198.025,Z 418.922,A -85,B 0,C 180,E1 -21826.868,E2 -21826.868} C_VEL
LIN {X 0,Y 204.082,Z 428.142,A -85,B 0,C 180,E1 -21828.875,E2 -21828.875} C_VEL
LIN {X 0,Y 208.059,Z 435.172,A -85,B 0,C 180,E1 -21830.142,E2 -21830.142} C_VEL
LIN {X 0,Y 214.354,Z 448.383,A -85,B 0,C 180,E1 -21832.095,E2 -21832.095} C_VEL
LIN {X 0,Y 219.189,Z 460.051,A -85,B 0,C 180,E1 -21833.548,E2 -21833.548} C_VEL
LIN {X 0,Y 217.171,Z 503.619,A -85,B 0,C 180,E1 -21834.899,E2 -21834.899} C_VEL
LIN {X 0,Y 216.203,Z 519.131,A -85,B 0,C 180,E1 -21835.497,E2 -21835.497} C_VEL
LIN {X 0,Y 214.64,Z 531.769,A -85,B 0,C 180,E1 -21836.318,E2 -21836.318} C_VEL
LIN {X 0,Y 212.533,Z 544.244,A -85,B 0,C 180,E1 -21837.497,E2 -21837.497} C_VEL
LIN {X 0,Y 210.045,Z 556.204,A -85,B 0,C 180,E1 -21839.04,E2 -21839.04} C_VEL
LIN {X 0,Y 207.288,Z 566.859,A -85,B 0,C 180,E1 -21840.832,E2 -21840.832} C_VEL
LIN {X 0,Y 204.454,Z 576.569,A -85,B 0,C 180,E1 -21842.906,E2 -21842.906} C_VEL
LIN {X 0,Y 201.704,Z 585.401,A -85,B 0,C 180,E1 -21845.284,E2 -21845.284} C_VEL
LIN {X 0,Y 199.225,Z 592.687,A -85,B 0,C 180,E1 -21847.715,E2 -21847.715} C_VEL
LIN {X 0,Y 196.527,Z 599.859,A -85,B 0,C 180,E1 -21850.684,E2 -21850.684} C_VEL
LIN {X 0,Y 194.702,Z 604.692,A -85,B 0,C 180,E1 -21853.216,E2 -21853.216} C_VEL
LIN {X 0,Y 192.927,Z 609.388,A -85,B 0,C 180,E1 -21856.303,E2 -21856.303} C_VEL
LIN {X 0,Y 191.66,Z 612.979,A -85,B 0,C 180,E1 -21859.436,E2 -21859.436} C_VEL
LIN {X 0,Y 191.062,Z 614.832,A -85,B 0,C 180,E1 -21861.539,E2 -21861.539} C_VEL
LIN {X 0,Y 190.405,Z 617.213,A -85,B 0,C 180,E1 -21865.767,E2 -21865.767} C_VEL
LIN {X 0,Y 190.269,Z 617.82,A -85,B 0,C 180,E1 -21867.884,E2 -21867.884} C_VEL
LIN {X 0,Y 190.236,Z 618.048,A -85,B 0,C 180,E1 -21870,E2 -21870} C_VEL
LIN {X 0,Y 190.269,Z 617.853,A -85,B 0,C 180,E1 -21872.117,E2 -21872.117} C_VEL
LIN {X 0,Y 190.46,Z 617.008,A -85,B 0,C 180,E1 -21874.925,E2 -21874.925} C_VEL
LIN {X 0,Y 191.066,Z 614.939,A -85,B 0,C 180,E1 -21878.461,E2 -21878.461} C_VEL
LIN {X 0,Y 192.018,Z 612.067,A -85,B 0,C 180,E1 -21881.614,E2 -21881.614} C_VEL
LIN {X 0,Y 193.43,Z 608.171,A -85,B 0,C 180,E1 -21884.735,E2 -21884.735} C_VEL
LIN {X 0,Y 195.282,Z 603.145,A -85,B 0,C 180,E1 -21887.813,E2 -21887.813} C_VEL
LIN {X 0,Y 197.728,Z 596.81,A -85,B 0,C 180,E1 -21890.821,E2 -21890.821} C_VEL
LIN {X 0,Y 200.617,Z 588.884,A -85,B 0,C 180,E1 -21893.758,E2 -21893.758} C_VEL
LIN {X 0,Y 203.444,Z 580.116,A -85,B 0,C 180,E1 -21896.348,E2 -21896.348} C_VEL
LIN {X 0,Y 206.175,Z 570.949,A -85,B 0,C 180,E1 -21898.505,E2 -21898.505} C_VEL
LIN {X 0,Y 209.236,Z 559.841,A -85,B 0,C 180,E1 -21900.533,E2 -21900.533} C_VEL
LIN {X 0,Y 211.755,Z 548.951,A -85,B 0,C 180,E1 -21902.076,E2 -21902.076} C_VEL
LIN {X 0,Y 214.011,Z 536.911,A -85,B 0,C 180,E1 -21903.372,E2 -21903.372} C_VEL
LIN {X 0,Y 215.76,Z 523.912,A -85,B 0,C 180,E1 -21904.374,E2 -21904.374} C_VEL
LIN {X 0,Y 216.964,Z 510.162,A -85,B 0,C 180,E1 -21905.023,E2 -21905.023} C_VEL
LIN {X 0,Y 219.374,Z 460.351,A -85,B 0,C 180,E1 -21906.561,E2 -21906.561} C_VEL
LIN {X 0,Y 213.563,Z 446.4,A -85,B 0,C 180,E1 -21908.317,E2 -21908.317} C_VEL
LIN {X 0,Y 206.697,Z 432.499,A -85,B 0,C 180,E1 -21910.465,E2 -21910.465} C_VEL
LIN {X 0,Y 202.732,Z 425.971,A -85,B 0,C 180,E1 -21911.736,E2 -21911.736} C_VEL
LIN {X 0,Y 197.873,Z 418.747,A -85,B 0,C 180,E1 -21913.364,E2 -21913.364} C_VEL
LIN {X 0,Y 195.686,Z 415.346,A -85,B 0,C 180,E1 -21914.145,E2 -21914.145} C_VEL
LIN {X 0,Y 193.276,Z 412.334,A -85,B 0,C 180,E1 -21915.001,E2 -21915.001} C_VEL
LIN {X 0,Y 192.566,Z 409.995,A -85,B 0,C 180,E1 -21915.354,E2 -21915.354} C_VEL
LIN {X 0,Y 192.548,Z 409.973,A -85,B 0,C 180,E1 -21920.041,E2 -21920.041} C_VEL
LIN {X 0,Y 192.602,Z 409.995,A -85,B 0,C 180,E1 -21924.279,E2 -21924.279} C_VEL
LIN {X 0,Y 192.611,Z 409.988,A -85,B 0,C 180,E1 -21929.28,E2 -21929.28} C_VEL
LIN {X 0,Y 192.668,Z 409.982,A -85,B 0,C 180,E1 -21931.692,E2 -21931.692} C_VEL
LIN {X 0,Y 192.716,Z 409.972,A -85,B 0,C 180,E1 -21936.35,E2 -21936.35} C_VEL
LIN {X 0,Y 192.786,Z 409.96,A -85,B 0,C 180,E1 -21941.413,E2 -21941.413} C_VEL
LIN {X 0,Y 192.858,Z 409.951,A -85,B 0,C 180,E1 -21947.37,E2 -21947.37} C_VEL
LIN {X 0,Y 193.077,Z 409.924,A -85,B 0,C 180,E1 -21951.628,E2 -21951.628} C_VEL
LIN {X 0,Y 193.269,Z 409.9,A -85,B 0,C 180,E1 -21957.916,E2 -21957.916} C_VEL
LIN {X 0,Y 193.448,Z 409.876,A -85,B 0,C 180,E1 -21960,E2 -21960} C_VEL
LIN {X 0,Y 192.977,Z 409.939,A -85,B 0,C 180,E1 -21964.177,E2 -21964.177} C_VEL
LIN {X 0,Y 193.038,Z 409.939,A -85,B 0,C 180,E1 -21968.374,E2 -21968.374} C_VEL
LIN {X 0,Y 192.806,Z 409.959,A -85,B 0,C 180,E1 -21972.633,E2 -21972.633} C_VEL
LIN {X 0,Y 192.762,Z 409.962,A -85,B 0,C 180,E1 -21976.958,E2 -21976.958} C_VEL
LIN {X 0,Y 192.64,Z 409.981,A -85,B 0,C 180,E1 -21981.397,E2 -21981.397} C_VEL
LIN {X 0,Y 192.668,Z 409.985,A -85,B 0,C 180,E1 -21984.224,E2 -21984.224} C_VEL
LIN {X 0,Y 192.647,Z 409.986,A -85,B 0,C 180,E1 -21988.889,E2 -21988.889} C_VEL
LIN {X 0,Y 192.599,Z 409.992,A -85,B 0,C 180,E1 -21993.186,E2 -21993.186} C_VEL
LIN {X 0,Y 192.554,Z 409.996,A -85,B 0,C 180,E1 -21998.351,E2 -21998.351} C_VEL
LIN {X 0,Y 192.564,Z 410.036,A -85,B 0,C 180,E1 -22002.066,E2 -22002.066} C_VEL
LIN {X 0,Y 193.717,Z 414.143,A -85,B 0,C 180,E1 -22004.936,E2 -22004.936} C_VEL
LIN {X 0,Y 196.02,Z 418.33,A -85,B 0,C 180,E1 -22005.813,E2 -22005.813} C_VEL
LIN {X 0,Y 197.546,Z 420.751,A -85,B 0,C 180,E1 -22006.359,E2 -22006.359} C_VEL
LIN {X 0,Y 203.424,Z 431.087,A -85,B 0,C 180,E1 -22008.389,E2 -22008.389} C_VEL
LIN {X 0,Y 208.843,Z 441.769,A -85,B 0,C 180,E1 -22010.159,E2 -22010.159} C_VEL
LIN {X 0,Y 214.515,Z 454.484,A -85,B 0,C 180,E1 -22011.936,E2 -22011.936} C_VEL
LIN {X 0,Y 217.704,Z 463.155,A -85,B 0,C 180,E1 -22012.938,E2 -22012.938} C_VEL
LIN {X 0,Y 218.186,Z 466.646,A -85,B 0,C 180,E1 -22013.174,E2 -22013.174} C_VEL
LIN {X 0,Y 217.932,Z 470.536,A -85,B 0,C 180,E1 -22013.28,E2 -22013.28} C_VEL
LIN {X 0,Y 215.705,Z 476.814,A -85,B 0,C 180,E1 -22013.096,E2 -22013.096} C_VEL
LIN {X 0,Y 213.147,Z 483.127,A -85,B 0,C 180,E1 -22012.842,E2 -22012.842} C_VEL
LIN {X 0,Y 212.411,Z 487.113,A -85,B 0,C 180,E1 -22012.858,E2 -22012.858} C_VEL
LIN {X 0,Y 210.457,Z 523.684,A -85,B 0,C 180,E1 -22014.062,E2 -22014.062} C_VEL
LIN {X 0,Y 208.789,Z 537.482,A -85,B 0,C 180,E1 -22014.858,E2 -22014.858} C_VEL
LIN {X 0,Y 206.799,Z 549.289,A -85,B 0,C 180,E1 -22015.892,E2 -22015.892} C_VEL
